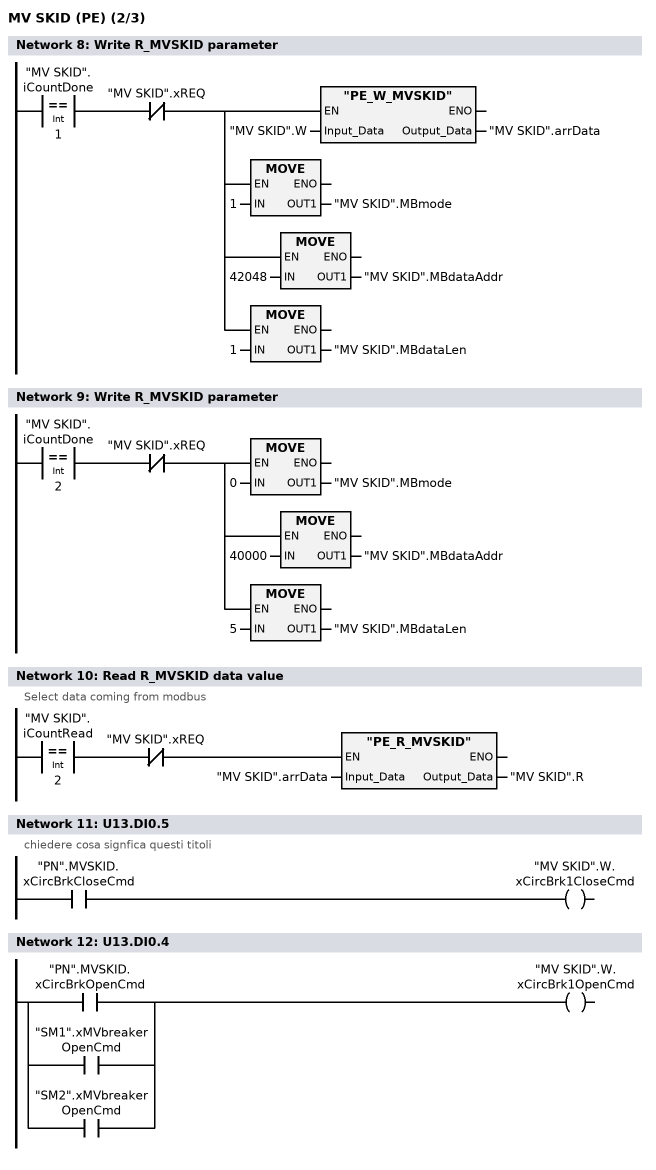
   RUNG wire#powerrail
      { S7_Templates := "SrcType := Int" } EQ_Contact(in1 := "MV SKID".iCountDone, in2 := 1)
      I_Contact( "MV SKID".xREQ )
      wire#w1
      "PE_W_MVSKID"(Input_Data := "MV SKID".W, Output_Data => "MV SKID".arrData)
   END_RUNG
   RUNG wire#w1
      Move(in := 1, out1 => "MV SKID".MBmode)
   END_RUNG
   RUNG wire#w1
      Move(in := 42048, out1 => "MV SKID".MBdataAddr)
   END_RUNG
   RUNG wire#w1
      Move(in := 1, out1 => "MV SKID".MBdataLen)
   END_RUNG
   // the same network as SCL:
   #_w1 := ("MV SKID".iCountDone = 1) AND NOT "MV SKID".xREQ;
   IF #_w1 THEN
       "PE_W_MVSKID"(Input_Data := "MV SKID".W, Output_Data => "MV SKID".arrData);
       "MV SKID".MBmode := 1;
       "MV SKID".MBdataAddr := 42048;
       "MV SKID".MBdataLen := 1;
   END_IF;
END_REGION

REGION Network 9: Write R_MVSKID parameter
   RUNG wire#powerrail
      { S7_Templates := "SrcType := Int" } EQ_Contact(in1 := "MV SKID".iCountDone, in2 := 2)
      I_Contact( "MV SKID".xREQ )
      wire#w1
      Move(in := 0, out1 => "MV SKID".MBmode)
   END_RUNG
   RUNG wire#w1
      Move(in := 40000, out1 => "MV SKID".MBdataAddr)
   END_RUNG
   RUNG wire#w1
      Move(in := 5, out1 => "MV SKID".MBdataLen)
   END_RUNG
   // the same network as SCL:
   IF ("MV SKID".iCountDone = 2) AND NOT "MV SKID".xREQ THEN
       "MV SKID".MBmode := 0;
       "MV SKID".MBdataAddr := 40000;
       "MV SKID".MBdataLen := 5;
   END_IF;
END_REGION

REGION Network 10: Read R_MVSKID data value
   // Select data coming from modbus
   RUNG wire#powerrail
      { S7_Templates := "SrcType := Int" } EQ_Contact(in1 := "MV SKID".iCountRead, in2 := 2)
      I_Contact( "MV SKID".xREQ )
      "PE_R_MVSKID"(Input_Data := "MV SKID".arrData, Output_Data => "MV SKID".R)
   END_RUNG
   // the same network as SCL:
   IF ("MV SKID".iCountRead = 2) AND NOT "MV SKID".xREQ THEN
       "PE_R_MVSKID"(Input_Data := "MV SKID".arrData, Output_Data => "MV SKID".R);
   END_IF;
END_REGION

REGION Network 11: U13.DI0.5
   // chiedere cosa signfica questi titoli
   RUNG wire#powerrail
      Contact( "PN".MVSKID.xCircBrkCloseCmd )
      Coil( "MV SKID".W.xCircBrk1CloseCmd )
   END_RUNG
   // the same network as SCL:
   "MV SKID".W.xCircBrk1CloseCmd := "PN".MVSKID.xCircBrkCloseCmd;
END_REGION

REGION Network 12: U13.DI0.4
   RUNG wire#powerrail
      Contact( "PN".MVSKID.xCircBrkOpenCmd )
      wire#w1
      Coil( "MV SKID".W.xCircBrk1OpenCmd )
   END_RUNG
   RUNG wire#powerrail
      Contact( "SM1".xMVbreakerOpenCmd )
   END_RUNG wire#w1
   RUNG wire#powerrail
      Contact( "SM2".xMVbreakerOpenCmd )
   END_RUNG wire#w1
   // the same network as SCL:
   "MV SKID".W.xCircBrk1OpenCmd := "PN".MVSKID.xCircBrkOpenCmd OR "SM1".xMVbreakerOpenCmd OR "SM2".xMVbreakerOpenCmd;
END_REGION

REGION Network 13: MV SKID Fault
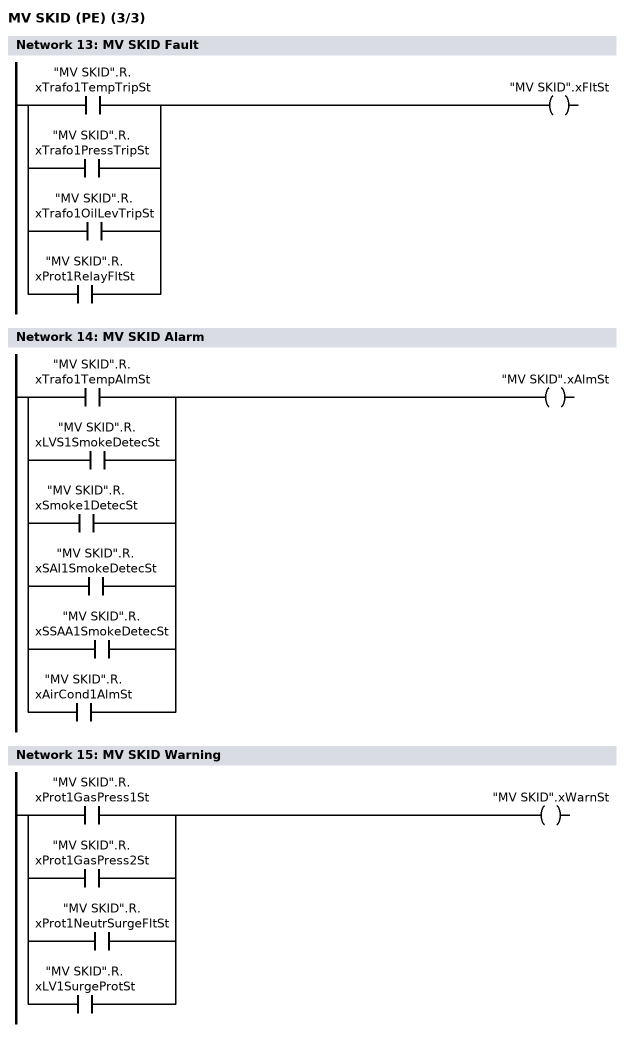
   RUNG wire#powerrail
      Contact( "MV SKID".R.xTrafo1TempTripSt )
      wire#w1
      Coil( "MV SKID".xFltSt )
   END_RUNG
   RUNG wire#powerrail
      Contact( "MV SKID".R.xTrafo1PressTripSt )
   END_RUNG wire#w1
   RUNG wire#powerrail
      Contact( "MV SKID".R.xTrafo1OilLevTripSt )
   END_RUNG wire#w1
   RUNG wire#powerrail
      Contact( "MV SKID".R.xProt1RelayFltSt )
   END_RUNG wire#w1
   // the same network as SCL:
   "MV SKID".xFltSt := "MV SKID".R.xTrafo1TempTripSt OR "MV SKID".R.xTrafo1PressTripSt OR "MV SKID".R.xTrafo1OilLevTripSt OR "MV SKID".R.xProt1RelayFltSt;
END_REGION

REGION Network 14: MV SKID Alarm
   RUNG wire#powerrail
      Contact( "MV SKID".R.xTrafo1TempAlmSt )
      wire#w1
      Coil( "MV SKID".xAlmSt )
   END_RUNG
   RUNG wire#powerrail
      Contact( "MV SKID".R.xLVS1SmokeDetecSt )
   END_RUNG wire#w1
   RUNG wire#powerrail
      Contact( "MV SKID".R.xSmoke1DetecSt )
   END_RUNG wire#w1
   RUNG wire#powerrail
      Contact( "MV SKID".R.xSAI1SmokeDetecSt )
   END_RUNG wire#w1
   RUNG wire#powerrail
      Contact( "MV SKID".R.xSSAA1SmokeDetecSt )
   END_RUNG wire#w1
   RUNG wire#powerrail
      Contact( "MV SKID".R.xAirCond1AlmSt )
   END_RUNG wire#w1
   // the same network as SCL:
   "MV SKID".xAlmSt := "MV SKID".R.xTrafo1TempAlmSt OR "MV SKID".R.xLVS1SmokeDetecSt OR "MV SKID".R.xSmoke1DetecSt OR "MV SKID".R.xSAI1SmokeDetecSt OR "MV SKID".R.xSSAA1SmokeDetecSt OR "MV SKID".R.xAirCond1AlmSt;
END_REGION

REGION Network 15: MV SKID Warning
   RUNG wire#powerrail
      Contact( "MV SKID".R.xProt1GasPress1St )
      wire#w1
      Coil( "MV SKID".xWarnSt )
   END_RUNG
   RUNG wire#powerrail
      Contact( "MV SKID".R.xProt1GasPress2St )
   END_RUNG wire#w1
   RUNG wire#powerrail
      Contact( "MV SKID".R.xProt1NeutrSurgeFltSt )
   END_RUNG wire#w1
   RUNG wire#powerrail
      Contact( "MV SKID".R.xLV1SurgeProtSt )
   END_RUNG wire#w1
   // the same network as SCL:
   "MV SKID".xWarnSt := "MV SKID".R.xProt1GasPress1St OR "MV SKID".R.xProt1GasPress2St OR "MV SKID".R.xProt1NeutrSurgeFltSt OR "MV SKID".R.xLV1SurgeProtSt;
END_REGION

REGION Network 16 (SCL): MV SKID Line Disconnector & Breaker Status
   "MV SKID".wLine1DiscSt.%X0 := "MV SKID".R.xLine1DiscOpenSt;
   "MV SKID".wLine1DiscSt.%X1 := "MV SKID".R.xLine1DiscCloseSt;
   "MV SKID".wLine1DiscSt.%X2 := "MV SKID".R.xLine1GndCloseSt;

   "MV SKID".wLine2DiscSt.%X0 := "MV SKID".R.xLine2DiscOpenSt;
   "MV SKID".wLine2DiscSt.%X1 := "MV SKID".R.xLine2DiscCloseSt;
   "MV SKID".wLine2DiscSt.%X2 := "MV SKID".R.xLine2GndCloseSt;

   "MV SKID".wProt1DiscSt.%X0 := "MV SKID".R.xProt1DiscOpenSt;
   "MV SKID".wProt1DiscSt.%X1 := "MV SKID".R.xProt1DiscCloseSt;
   "MV SKID".wProt1DiscSt.%X2 := "MV SKID".R.xProt1GndCloseSt;

   "MV SKID".wProt1CircBrkSt.%X0 := "MV SKID".R.xProt1CircBrkOpenSt;
   "MV SKID".wProt1CircBrkSt.%X1 := "MV SKID".R.xProt1CircBrkCloseSt;
END_REGION
END_FUNCTION

FUNCTION "PE_W_MVSKID" : Void
{ S7_Optimized_Access := 'TRUE' }
VERSION : 0.1
   VAR_INPUT 
      Input_Data : "W_MV";
   END_VAR

   VAR_OUTPUT 
      Output_Data : Array[1..125] of Word;
   END_VAR


BEGIN
	REGION
	    // 2022/01/24
	END_REGION
	
	REGION
	    
	    #Output_Data[1].%X0 := #Input_Data.xCircBrk1OpenCmd;
	    #Output_Data[1].%X1 := #Input_Data.xCircBrk1CloseCmd;
	    #Output_Data[1].%X2 := #Input_Data.xLVCircBrk1OpenCmd;
	    #Output_Data[1].%X3 := #Input_Data.xLVCircBrk1CloseCmd;
	    #Output_Data[1].%X4 := #Input_Data.xCircBrk2OpenCmd;
	    #Output_Data[1].%X5 := #Input_Data.xCircBrk2CloseCmd;
	    #Output_Data[1].%X6 := #Input_Data.xLVCircBrk2OpenCmd;
	    #Output_Data[1].%X7 := #Input_Data.xLVCircBrk2CloseCmd;
	    
	END_REGION
END_FUNCTION

FUNCTION "PE_R_MVSKID" : Void
{ S7_Optimized_Access := 'TRUE' }
VERSION : 0.1
   VAR_INPUT 
      Input_Data : Array[1..125] of Word;
   END_VAR

   VAR_OUTPUT 
      Output_Data : "R_MV";
   END_VAR


BEGIN
	REGION
	    // 2022/01/24
	END_REGION
	
	REGION
	    
	    #Output_Data.xTrafo1TempTripSt      := #Input_Data[1].%X0;
	    #Output_Data.xTrafo1TempAlmSt       := #Input_Data[1].%X1;
	    #Output_Data.xTrafo1PressTripSt     := #Input_Data[1].%X2;
	    #Output_Data.xTrafo1OilLevTripSt    := #Input_Data[1].%X3;
	    #Output_Data.xLine1DiscOpenSt       := #Input_Data[1].%X4;
	    #Output_Data.xLine1DiscCloseSt      := #Input_Data[1].%X5;
	    #Output_Data.xLine1GndCloseSt       := #Input_Data[1].%X6;
	    #Output_Data.xProt1GasPress1St      := #Input_Data[1].%X7;
	    
	    #Output_Data.xLine2DiscOpenSt       := #Input_Data[1].%X8;
	    #Output_Data.xLine2DiscCloseSt      := #Input_Data[1].%X9;
	    #Output_Data.xLine2GndCloseSt       := #Input_Data[1].%X10;
	    #Output_Data.xProt1DiscCloseSt      := #Input_Data[1].%X11;
	    #Output_Data.xProt1DiscOpenSt       := #Input_Data[1].%X12;
	    #Output_Data.xProt1GndCloseSt       := #Input_Data[1].%X13;
	    #Output_Data.xProt1CircBrkOpenSt    := #Input_Data[1].%X14;
	    #Output_Data.xProt1CircBrkCloseSt   := #Input_Data[1].%X15;
	    
	    #Output_Data.xProt1RelayFltSt       := #Input_Data[2].%X0;
	    #Output_Data.xLV1SurgeProtSt        := #Input_Data[2].%X1;
	    #Output_Data.xSpring1ChargeSt       := #Input_Data[2].%X2;
	    #Output_Data.xProt1GasPress2St      := #Input_Data[2].%X3;
	    #Output_Data.xBackfeedtrakers1St    := #Input_Data[2].%X4;
	    #Output_Data.xProt1NeutrSurgeFltSt  := #Input_Data[2].%X5;
	    #Output_Data.xLVS1SmokeDetecSt       := #Input_Data[2].%X6;
	    #Output_Data.xSmoke1DetecSt         := #Input_Data[2].%X7;
	    
	    #Output_Data.xSAI1SmokeDetecSt      := #Input_Data[2].%X8;
	    #Output_Data.xSSAA1SmokeDetecSt     := #Input_Data[2].%X9;
	    #Output_Data.xAirCond1AlmSt         := #Input_Data[2].%X10;
	    #Output_Data.xAcBrkHENK1OpenSt      := #Input_Data[2].%X11;
	    #Output_Data.xAcBrkHENK1CloseSt     := #Input_Data[2].%X12;
	    #Output_Data.xTrafo2TempTripSt      := #Input_Data[2].%X13;
	    #Output_Data.xTrafo2TempAlmSt       := #Input_Data[2].%X14;
	    #Output_Data.xTrafo2PressTripSt     := #Input_Data[2].%X15;
	    
	    #Output_Data.xTrafo2OilLevTripSt    := #Input_Data[3].%X0;
	    #Output_Data.xProt2DiscCloseSt      := #Input_Data[3].%X1;
	    #Output_Data.xProt2DiscOpenSt       := #Input_Data[3].%X2;
	    #Output_Data.xProt2GndCloseSt       := #Input_Data[3].%X3;
	    #Output_Data.xProt2CircBrkOpenSt    := #Input_Data[3].%X4;
	    #Output_Data.xProt2CircBrkCloseSt   := #Input_Data[3].%X5;
	    #Output_Data.xProt2NCWatchdogSt     := #Input_Data[3].%X6;
	    #Output_Data.xLV2SurgeProtSt        := #Input_Data[3].%X7;
	    
	    #Output_Data.xSpring2ChargeSt       := #Input_Data[3].%X8;
	    #Output_Data.xAcBrkHENK2OpenSt      := #Input_Data[3].%X9;
	    #Output_Data.xAcBrkHENK2CloseSt     := #Input_Data[3].%X10;
	    #Output_Data.xBackfeedtrakers2St    := #Input_Data[3].%X11;
	    #Output_Data.xProt2NeutrSurgeSt     := #Input_Data[3].%X12;
	    #Output_Data.xSAI2SmokeDetecSt      := #Input_Data[3].%X13;
	    #Output_Data.xSSAA2SmokeDetecSt     := #Input_Data[3].%X14;
	    #Output_Data.xAirCond2AlmSt         := #Input_Data[3].%X15;
	    
	    #Output_Data.rPT100Trafo1St         := INT_TO_REAL(WORD_TO_INT(#Input_Data[4]))/10.0;
	    #Output_Data.rPT100Trafo2St         := INT_TO_REAL(WORD_TO_INT(#Input_Data[5]))/10.0;
	    
	END_REGION
END_FUNCTION

FUNCTION "PCS1 Faults" : Void   // FC43, LAD
{ S7_Optimized_Access := 'TRUE' }
VERSION : 0.1
// stored: AutoNumber false, IsIECCheckEnabled false, SetENOAutomatically false, UDAEnableTagReadback false
   VAR_TEMP
      wMF1 : Word;
      wMF2 : Word;
      wMF3 : Word;
      wMF4 : Word;
      wMW1 : Word;
      wMW2 : Word;
      wMW3 : Word;
      wMW4 : Word;
   END_VAR
   VAR_TEMP   // added for the SCL form of the ladder/FBD networks
      _w1 : Bool;
      _w2 : Bool;
      _w3 : Bool;
      _w4 : Bool;
   END_VAR
BEGIN

REGION Network 1: Split Inverter fault & warning and Module number
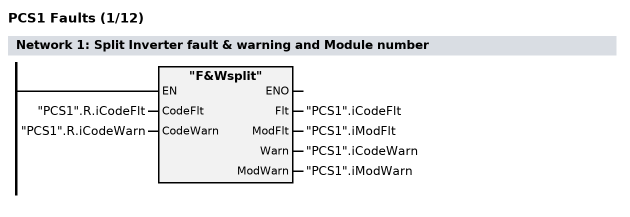
   RUNG wire#powerrail
      "F&Wsplit"(CodeFlt := "PCS1".R.iCodeFlt, CodeWarn := "PCS1".R.iCodeWarn, Flt => "PCS1".iCodeFlt, ModFlt => "PCS1".iModFlt, Warn => "PCS1".iCodeWarn, ModWarn => "PCS1".iModWarn)
   END_RUNG
   // the same network as SCL:
   "F&Wsplit"(CodeFlt := "PCS1".R.iCodeFlt,
              CodeWarn := "PCS1".R.iCodeWarn,
              Flt => "PCS1".iCodeFlt,
              ModFlt => "PCS1".iModFlt,
              Warn => "PCS1".iCodeWarn,
              ModWarn => "PCS1".iModWarn);
END_REGION

REGION Network 2: Inverter Faults
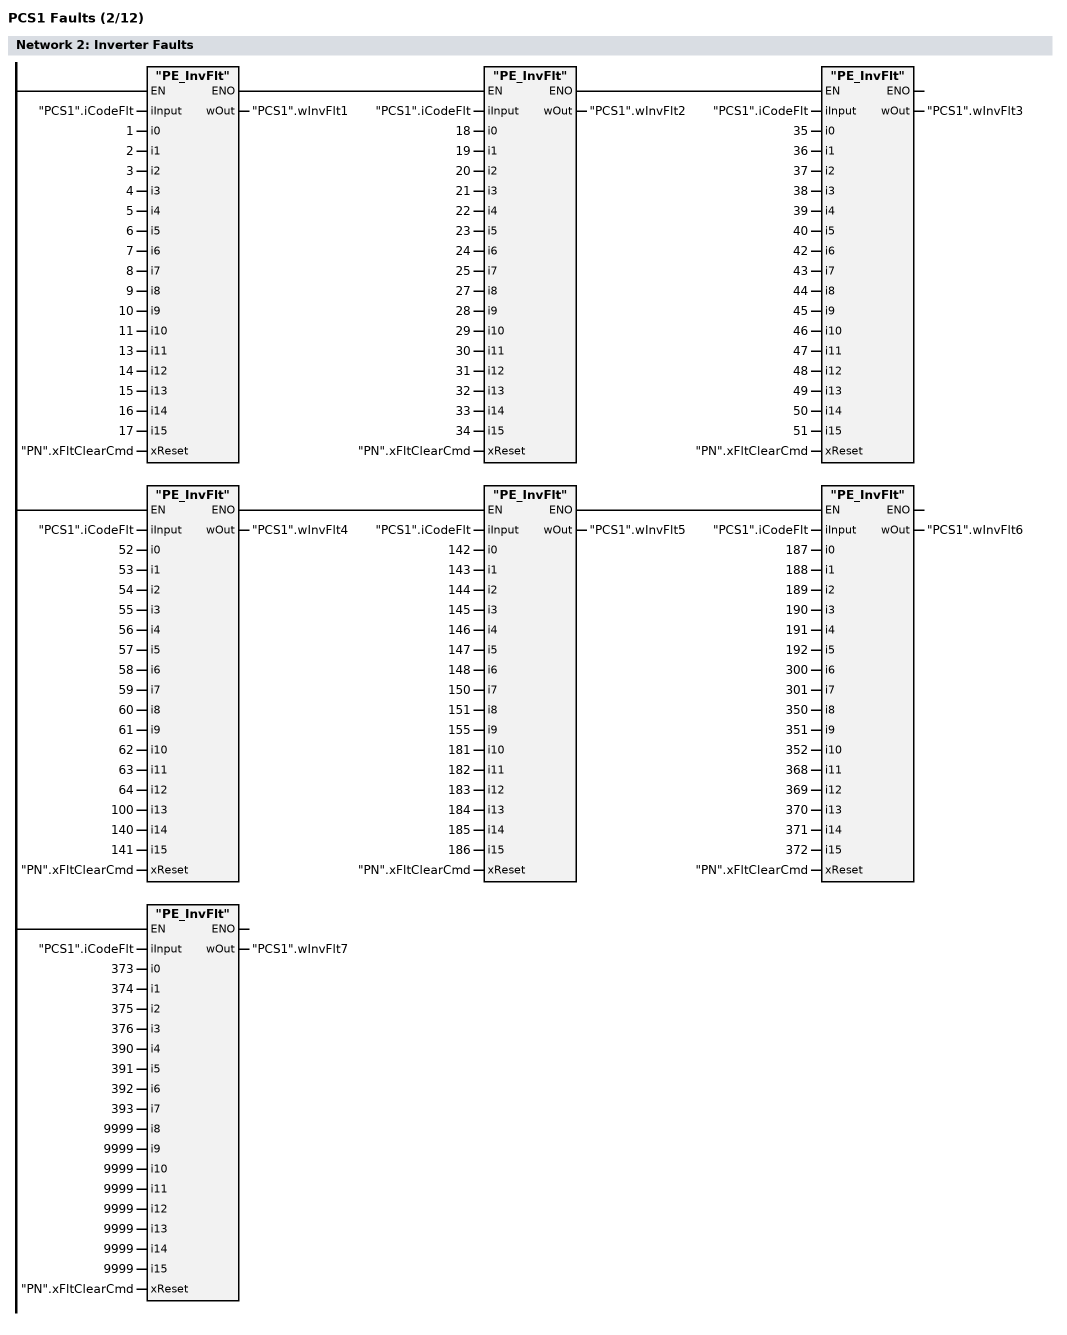
   RUNG wire#powerrail
      "PE_InvFlt"(iInput := "PCS1".iCodeFlt, i0 := 1, i1 := 2, i2 := 3, i3 := 4, i4 := 5, i5 := 6, i6 := 7, i7 := 8, i8 := 9, i9 := 10, i10 := 11, i11 := 13, i12 := 14, i13 := 15, i14 := 16, i15 := 17, xReset := "PN".xFltClearCmd, wOut => "PCS1".wInvFlt1)
      "PE_InvFlt"(iInput := "PCS1".iCodeFlt, i0 := 18, i1 := 19, i2 := 20, i3 := 21, i4 := 22, i5 := 23, i6 := 24, i7 := 25, i8 := 27, i9 := 28, i10 := 29, i11 := 30, i12 := 31, i13 := 32, i14 := 33, i15 := 34, xReset := "PN".xFltClearCmd, wOut => "PCS1".wInvFlt2)
      "PE_InvFlt"(iInput := "PCS1".iCodeFlt, i0 := 35, i1 := 36, i2 := 37, i3 := 38, i4 := 39, i5 := 40, i6 := 42, i7 := 43, i8 := 44, i9 := 45, i10 := 46, i11 := 47, i12 := 48, i13 := 49, i14 := 50, i15 := 51, xReset := "PN".xFltClearCmd, wOut => "PCS1".wInvFlt3)
   END_RUNG
   RUNG wire#powerrail
      "PE_InvFlt"(iInput := "PCS1".iCodeFlt, i0 := 52, i1 := 53, i2 := 54, i3 := 55, i4 := 56, i5 := 57, i6 := 58, i7 := 59, i8 := 60, i9 := 61, i10 := 62, i11 := 63, i12 := 64, i13 := 100, i14 := 140, i15 := 141, xReset := "PN".xFltClearCmd, wOut => "PCS1".wInvFlt4)
      "PE_InvFlt"(iInput := "PCS1".iCodeFlt, i0 := 142, i1 := 143, i2 := 144, i3 := 145, i4 := 146, i5 := 147, i6 := 148, i7 := 150, i8 := 151, i9 := 155, i10 := 181, i11 := 182, i12 := 183, i13 := 184, i14 := 185, i15 := 186, xReset := "PN".xFltClearCmd, wOut => "PCS1".wInvFlt5)
      "PE_InvFlt"(iInput := "PCS1".iCodeFlt, i0 := 187, i1 := 188, i2 := 189, i3 := 190, i4 := 191, i5 := 192, i6 := 300, i7 := 301, i8 := 350, i9 := 351, i10 := 352, i11 := 368, i12 := 369, i13 := 370, i14 := 371, i15 := 372, xReset := "PN".xFltClearCmd, wOut => "PCS1".wInvFlt6)
   END_RUNG
   RUNG wire#powerrail
      "PE_InvFlt"(iInput := "PCS1".iCodeFlt, i0 := 373, i1 := 374, i2 := 375, i3 := 376, i4 := 390, i5 := 391, i6 := 392, i7 := 393, i8 := 9999, i9 := 9999, i10 := 9999, i11 := 9999, i12 := 9999, i13 := 9999, i14 := 9999, i15 := 9999, xReset := "PN".xFltClearCmd, wOut => "PCS1".wInvFlt7)
   END_RUNG
   // the same network as SCL:
   "PE_InvFlt"(iInput := "PCS1".iCodeFlt,
               i0 := 1,
               i1 := 2,
               i2 := 3,
               i3 := 4,
               i4 := 5,
               i5 := 6,
               i6 := 7,
               i7 := 8,
               i8 := 9,
               i9 := 10,
               i10 := 11,
               i11 := 13,
               i12 := 14,
               i13 := 15,
               i14 := 16,
               i15 := 17,
               xReset := "PN".xFltClearCmd,
               wOut => "PCS1".wInvFlt1,
               ENO => #_w1);
   "PE_InvFlt"(EN := #_w1,
               iInput := "PCS1".iCodeFlt,
               i0 := 18,
               i1 := 19,
               i2 := 20,
               i3 := 21,
               i4 := 22,
               i5 := 23,
               i6 := 24,
               i7 := 25,
               i8 := 27,
               i9 := 28,
               i10 := 29,
               i11 := 30,
               i12 := 31,
               i13 := 32,
               i14 := 33,
               i15 := 34,
               xReset := "PN".xFltClearCmd,
               wOut => "PCS1".wInvFlt2,
               ENO => #_w2);
   IF #_w2 THEN
       "PE_InvFlt"(iInput := "PCS1".iCodeFlt,
                   i0 := 35,
                   i1 := 36,
                   i2 := 37,
                   i3 := 38,
                   i4 := 39,
                   i5 := 40,
                   i6 := 42,
                   i7 := 43,
                   i8 := 44,
                   i9 := 45,
                   i10 := 46,
                   i11 := 47,
                   i12 := 48,
                   i13 := 49,
                   i14 := 50,
                   i15 := 51,
                   xReset := "PN".xFltClearCmd,
                   wOut => "PCS1".wInvFlt3);
   END_IF;
   "PE_InvFlt"(iInput := "PCS1".iCodeFlt,
               i0 := 52,
               i1 := 53,
               i2 := 54,
               i3 := 55,
               i4 := 56,
               i5 := 57,
               i6 := 58,
               i7 := 59,
               i8 := 60,
               i9 := 61,
               i10 := 62,
               i11 := 63,
               i12 := 64,
               i13 := 100,
               i14 := 140,
               i15 := 141,
               xReset := "PN".xFltClearCmd,
               wOut => "PCS1".wInvFlt4,
               ENO => #_w3);
   "PE_InvFlt"(EN := #_w3,
               iInput := "PCS1".iCodeFlt,
               i0 := 142,
               i1 := 143,
               i2 := 144,
               i3 := 145,
               i4 := 146,
               i5 := 147,
               i6 := 148,
               i7 := 150,
               i8 := 151,
               i9 := 155,
               i10 := 181,
               i11 := 182,
               i12 := 183,
               i13 := 184,
               i14 := 185,
               i15 := 186,
               xReset := "PN".xFltClearCmd,
               wOut => "PCS1".wInvFlt5,
               ENO => #_w4);
   IF #_w4 THEN
       "PE_InvFlt"(iInput := "PCS1".iCodeFlt,
                   i0 := 187,
                   i1 := 188,
                   i2 := 189,
                   i3 := 190,
                   i4 := 191,
                   i5 := 192,
                   i6 := 300,
                   i7 := 301,
                   i8 := 350,
                   i9 := 351,
                   i10 := 352,
                   i11 := 368,
                   i12 := 369,
                   i13 := 370,
                   i14 := 371,
                   i15 := 372,
                   xReset := "PN".xFltClearCmd,
                   wOut => "PCS1".wInvFlt6);
   END_IF;
   "PE_InvFlt"(iInput := "PCS1".iCodeFlt,
               i0 := 373,
               i1 := 374,
               i2 := 375,
               i3 := 376,
               i4 := 390,
               i5 := 391,
               i6 := 392,
               i7 := 393,
               i8 := 9999,
               i9 := 9999,
               i10 := 9999,
               i11 := 9999,
               i12 := 9999,
               i13 := 9999,
               i14 := 9999,
               i15 := 9999,
               xReset := "PN".xFltClearCmd,
               wOut => "PCS1".wInvFlt7);
END_REGION

REGION Network 3: Inverter Warning
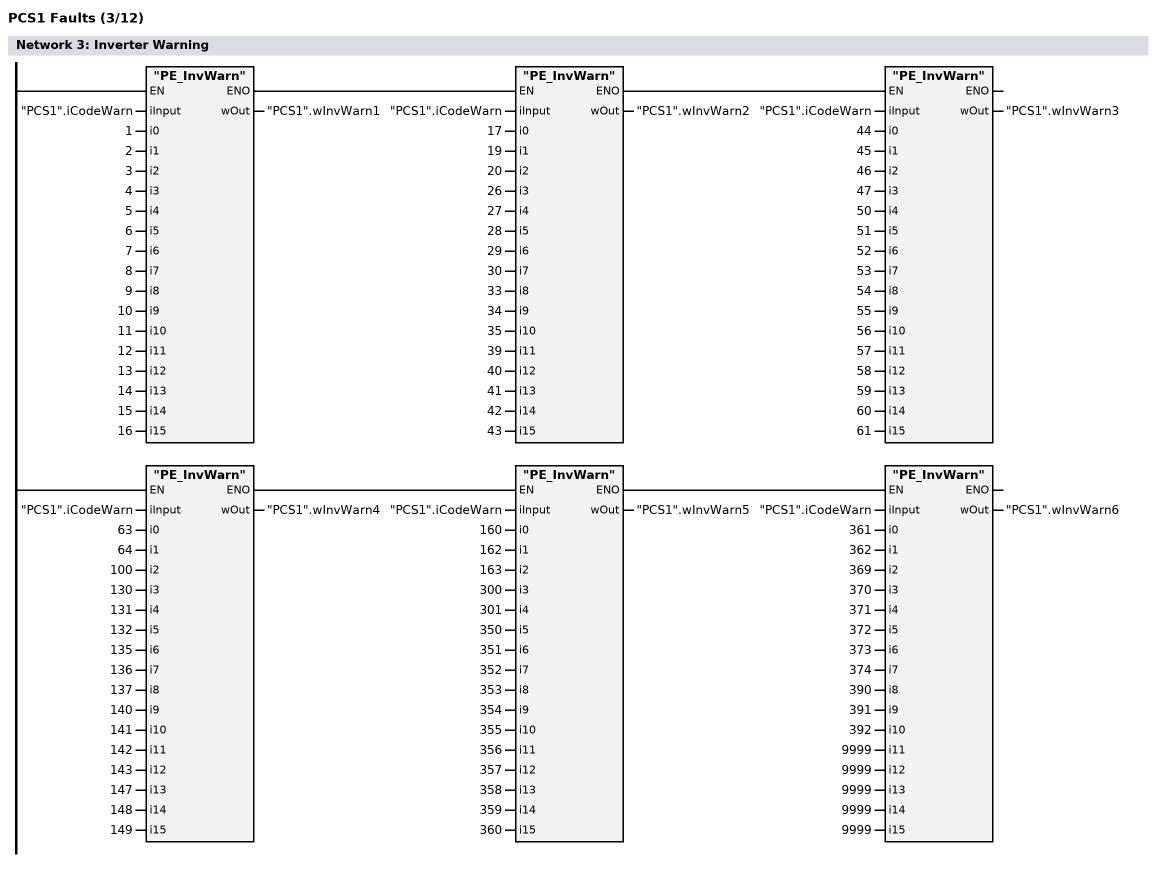
   RUNG wire#powerrail
      "PE_InvWarn"(iInput := "PCS1".iCodeWarn, i0 := 1, i1 := 2, i2 := 3, i3 := 4, i4 := 5, i5 := 6, i6 := 7, i7 := 8, i8 := 9, i9 := 10, i10 := 11, i11 := 12, i12 := 13, i13 := 14, i14 := 15, i15 := 16, wOut => "PCS1".wInvWarn1)
      "PE_InvWarn"(iInput := "PCS1".iCodeWarn, i0 := 17, i1 := 19, i2 := 20, i3 := 26, i4 := 27, i5 := 28, i6 := 29, i7 := 30, i8 := 33, i9 := 34, i10 := 35, i11 := 39, i12 := 40, i13 := 41, i14 := 42, i15 := 43, wOut => "PCS1".wInvWarn2)
      "PE_InvWarn"(iInput := "PCS1".iCodeWarn, i0 := 44, i1 := 45, i2 := 46, i3 := 47, i4 := 50, i5 := 51, i6 := 52, i7 := 53, i8 := 54, i9 := 55, i10 := 56, i11 := 57, i12 := 58, i13 := 59, i14 := 60, i15 := 61, wOut => "PCS1".wInvWarn3)
   END_RUNG
   RUNG wire#powerrail
      "PE_InvWarn"(iInput := "PCS1".iCodeWarn, i0 := 63, i1 := 64, i2 := 100, i3 := 130, i4 := 131, i5 := 132, i6 := 135, i7 := 136, i8 := 137, i9 := 140, i10 := 141, i11 := 142, i12 := 143, i13 := 147, i14 := 148, i15 := 149, wOut => "PCS1".wInvWarn4)
      "PE_InvWarn"(iInput := "PCS1".iCodeWarn, i0 := 160, i1 := 162, i2 := 163, i3 := 300, i4 := 301, i5 := 350, i6 := 351, i7 := 352, i8 := 353, i9 := 354, i10 := 355, i11 := 356, i12 := 357, i13 := 358, i14 := 359, i15 := 360, wOut => "PCS1".wInvWarn5)
      "PE_InvWarn"(iInput := "PCS1".iCodeWarn, i0 := 361, i1 := 362, i2 := 369, i3 := 370, i4 := 371, i5 := 372, i6 := 373, i7 := 374, i8 := 390, i9 := 391, i10 := 392, i11 := 9999, i12 := 9999, i13 := 9999, i14 := 9999, i15 := 9999, wOut => "PCS1".wInvWarn6)
   END_RUNG
   // the same network as SCL:
   "PE_InvWarn"(iInput := "PCS1".iCodeWarn,
                i0 := 1,
                i1 := 2,
                i2 := 3,
                i3 := 4,
                i4 := 5,
                i5 := 6,
                i6 := 7,
                i7 := 8,
                i8 := 9,
                i9 := 10,
                i10 := 11,
                i11 := 12,
                i12 := 13,
                i13 := 14,
                i14 := 15,
                i15 := 16,
                wOut => "PCS1".wInvWarn1,
                ENO => #_w1);
   "PE_InvWarn"(EN := #_w1,
                iInput := "PCS1".iCodeWarn,
                i0 := 17,
                i1 := 19,
                i2 := 20,
                i3 := 26,
                i4 := 27,
                i5 := 28,
                i6 := 29,
                i7 := 30,
                i8 := 33,
                i9 := 34,
                i10 := 35,
                i11 := 39,
                i12 := 40,
                i13 := 41,
                i14 := 42,
                i15 := 43,
                wOut => "PCS1".wInvWarn2,
                ENO => #_w2);
   IF #_w2 THEN
       "PE_InvWarn"(iInput := "PCS1".iCodeWarn,
                    i0 := 44,
                    i1 := 45,
                    i2 := 46,
                    i3 := 47,
                    i4 := 50,
                    i5 := 51,
                    i6 := 52,
                    i7 := 53,
                    i8 := 54,
                    i9 := 55,
                    i10 := 56,
                    i11 := 57,
                    i12 := 58,
                    i13 := 59,
                    i14 := 60,
                    i15 := 61,
                    wOut => "PCS1".wInvWarn3);
   END_IF;
   "PE_InvWarn"(iInput := "PCS1".iCodeWarn,
                i0 := 63,
                i1 := 64,
                i2 := 100,
                i3 := 130,
                i4 := 131,
                i5 := 132,
                i6 := 135,
                i7 := 136,
                i8 := 137,
                i9 := 140,
                i10 := 141,
                i11 := 142,
                i12 := 143,
                i13 := 147,
                i14 := 148,
                i15 := 149,
                wOut => "PCS1".wInvWarn4,
                ENO => #_w3);
   "PE_InvWarn"(EN := #_w3,
                iInput := "PCS1".iCodeWarn,
                i0 := 160,
                i1 := 162,
                i2 := 163,
                i3 := 300,
                i4 := 301,
                i5 := 350,
                i6 := 351,
                i7 := 352,
                i8 := 353,
                i9 := 354,
                i10 := 355,
                i11 := 356,
                i12 := 357,
                i13 := 358,
                i14 := 359,
                i15 := 360,
                wOut => "PCS1".wInvWarn5,
                ENO => #_w4);
   IF #_w4 THEN
       "PE_InvWarn"(iInput := "PCS1".iCodeWarn,
                    i0 := 361,
                    i1 := 362,
                    i2 := 369,
                    i3 := 370,
                    i4 := 371,
                    i5 := 372,
                    i6 := 373,
                    i7 := 374,
                    i8 := 390,
                    i9 := 391,
                    i10 := 392,
                    i11 := 9999,
                    i12 := 9999,
                    i13 := 9999,
                    i14 := 9999,
                    i15 := 9999,
                    wOut => "PCS1".wInvWarn6);
   END_IF;
END_REGION

REGION Network 4: Module Faults
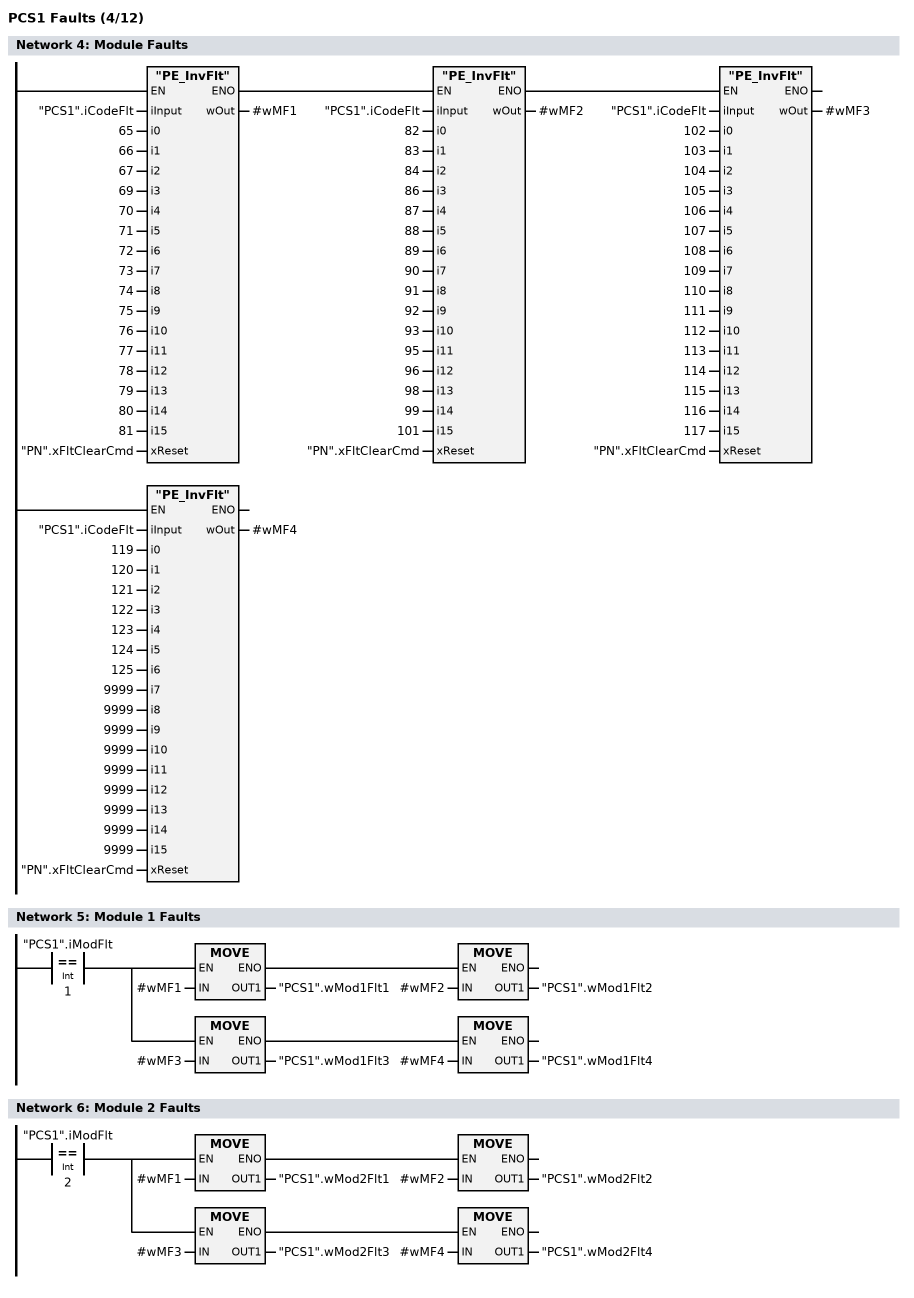
   RUNG wire#powerrail
      "PE_InvFlt"(iInput := "PCS1".iCodeFlt, i0 := 65, i1 := 66, i2 := 67, i3 := 69, i4 := 70, i5 := 71, i6 := 72, i7 := 73, i8 := 74, i9 := 75, i10 := 76, i11 := 77, i12 := 78, i13 := 79, i14 := 80, i15 := 81, xReset := "PN".xFltClearCmd, wOut => #wMF1)
      "PE_InvFlt"(iInput := "PCS1".iCodeFlt, i0 := 82, i1 := 83, i2 := 84, i3 := 86, i4 := 87, i5 := 88, i6 := 89, i7 := 90, i8 := 91, i9 := 92, i10 := 93, i11 := 95, i12 := 96, i13 := 98, i14 := 99, i15 := 101, xReset := "PN".xFltClearCmd, wOut => #wMF2)
      "PE_InvFlt"(iInput := "PCS1".iCodeFlt, i0 := 102, i1 := 103, i2 := 104, i3 := 105, i4 := 106, i5 := 107, i6 := 108, i7 := 109, i8 := 110, i9 := 111, i10 := 112, i11 := 113, i12 := 114, i13 := 115, i14 := 116, i15 := 117, xReset := "PN".xFltClearCmd, wOut => #wMF3)
   END_RUNG
   RUNG wire#powerrail
      "PE_InvFlt"(iInput := "PCS1".iCodeFlt, i0 := 119, i1 := 120, i2 := 121, i3 := 122, i4 := 123, i5 := 124, i6 := 125, i7 := 9999, i8 := 9999, i9 := 9999, i10 := 9999, i11 := 9999, i12 := 9999, i13 := 9999, i14 := 9999, i15 := 9999, xReset := "PN".xFltClearCmd, wOut => #wMF4)
   END_RUNG
   // the same network as SCL:
   "PE_InvFlt"(iInput := "PCS1".iCodeFlt,
               i0 := 65,
               i1 := 66,
               i2 := 67,
               i3 := 69,
               i4 := 70,
               i5 := 71,
               i6 := 72,
               i7 := 73,
               i8 := 74,
               i9 := 75,
               i10 := 76,
               i11 := 77,
               i12 := 78,
               i13 := 79,
               i14 := 80,
               i15 := 81,
               xReset := "PN".xFltClearCmd,
               wOut => #wMF1,
               ENO => #_w1);
   "PE_InvFlt"(EN := #_w1,
               iInput := "PCS1".iCodeFlt,
               i0 := 82,
               i1 := 83,
               i2 := 84,
               i3 := 86,
               i4 := 87,
               i5 := 88,
               i6 := 89,
               i7 := 90,
               i8 := 91,
               i9 := 92,
               i10 := 93,
               i11 := 95,
               i12 := 96,
               i13 := 98,
               i14 := 99,
               i15 := 101,
               xReset := "PN".xFltClearCmd,
               wOut => #wMF2,
               ENO => #_w2);
   IF #_w2 THEN
       "PE_InvFlt"(iInput := "PCS1".iCodeFlt,
                   i0 := 102,
                   i1 := 103,
                   i2 := 104,
                   i3 := 105,
                   i4 := 106,
                   i5 := 107,
                   i6 := 108,
                   i7 := 109,
                   i8 := 110,
                   i9 := 111,
                   i10 := 112,
                   i11 := 113,
                   i12 := 114,
                   i13 := 115,
                   i14 := 116,
                   i15 := 117,
                   xReset := "PN".xFltClearCmd,
                   wOut => #wMF3);
   END_IF;
   "PE_InvFlt"(iInput := "PCS1".iCodeFlt,
               i0 := 119,
               i1 := 120,
               i2 := 121,
               i3 := 122,
               i4 := 123,
               i5 := 124,
               i6 := 125,
               i7 := 9999,
               i8 := 9999,
               i9 := 9999,
               i10 := 9999,
               i11 := 9999,
               i12 := 9999,
               i13 := 9999,
               i14 := 9999,
               i15 := 9999,
               xReset := "PN".xFltClearCmd,
               wOut => #wMF4);
END_REGION

REGION Network 5: Module 1 Faults
   RUNG wire#powerrail
      { S7_Templates := "SrcType := Int" } EQ_Contact(in1 := "PCS1".iModFlt, in2 := 1)
      wire#w1
      Move(in := #wMF1, out1 => "PCS1".wMod1Flt1)
      Move(in := #wMF2, out1 => "PCS1".wMod1Flt2)
   END_RUNG
   RUNG wire#w1
      Move(in := #wMF3, out1 => "PCS1".wMod1Flt3)
      Move(in := #wMF4, out1 => "PCS1".wMod1Flt4)
   END_RUNG
   // the same network as SCL:
   IF "PCS1".iModFlt = 1 THEN
       "PCS1".wMod1Flt1 := #wMF1;
       "PCS1".wMod1Flt2 := #wMF2;
       "PCS1".wMod1Flt3 := #wMF3;
       "PCS1".wMod1Flt4 := #wMF4;
   END_IF;
END_REGION

REGION Network 6: Module 2 Faults
   RUNG wire#powerrail
      { S7_Templates := "SrcType := Int" } EQ_Contact(in1 := "PCS1".iModFlt, in2 := 2)
      wire#w1
      Move(in := #wMF1, out1 => "PCS1".wMod2Flt1)
      Move(in := #wMF2, out1 => "PCS1".wMod2Flt2)
   END_RUNG
   RUNG wire#w1
      Move(in := #wMF3, out1 => "PCS1".wMod2Flt3)
      Move(in := #wMF4, out1 => "PCS1".wMod2Flt4)
   END_RUNG
   // the same network as SCL:
   IF "PCS1".iModFlt = 2 THEN
       "PCS1".wMod2Flt1 := #wMF1;
       "PCS1".wMod2Flt2 := #wMF2;
       "PCS1".wMod2Flt3 := #wMF3;
       "PCS1".wMod2Flt4 := #wMF4;
   END_IF;
END_REGION

REGION Network 7: Module 3 Faults
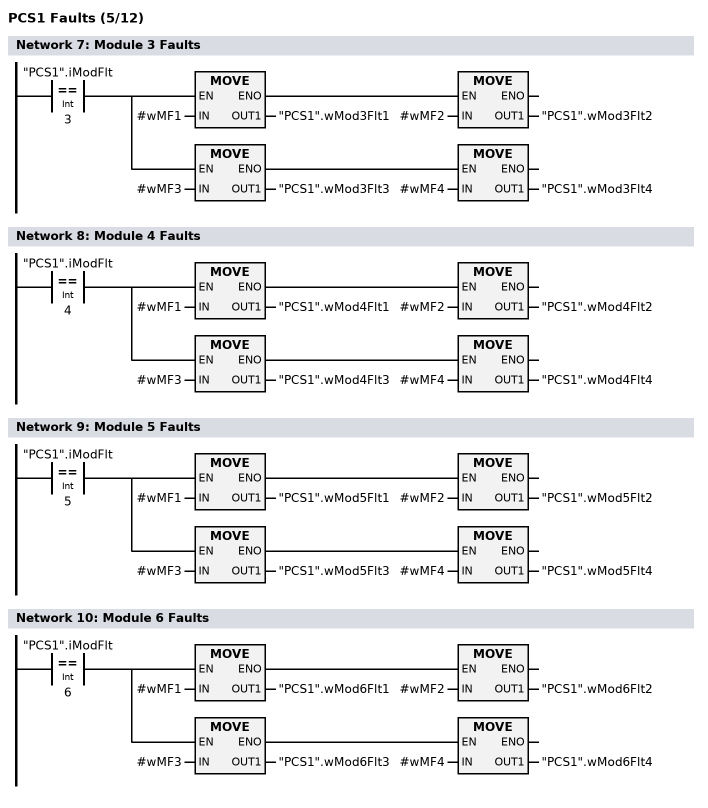
   RUNG wire#powerrail
      { S7_Templates := "SrcType := Int" } EQ_Contact(in1 := "PCS1".iModFlt, in2 := 3)
      wire#w1
      Move(in := #wMF1, out1 => "PCS1".wMod3Flt1)
      Move(in := #wMF2, out1 => "PCS1".wMod3Flt2)
   END_RUNG
   RUNG wire#w1
      Move(in := #wMF3, out1 => "PCS1".wMod3Flt3)
      Move(in := #wMF4, out1 => "PCS1".wMod3Flt4)
   END_RUNG
   // the same network as SCL:
   IF "PCS1".iModFlt = 3 THEN
       "PCS1".wMod3Flt1 := #wMF1;
       "PCS1".wMod3Flt2 := #wMF2;
       "PCS1".wMod3Flt3 := #wMF3;
       "PCS1".wMod3Flt4 := #wMF4;
   END_IF;
END_REGION

REGION Network 8: Module 4 Faults
   RUNG wire#powerrail
      { S7_Templates := "SrcType := Int" } EQ_Contact(in1 := "PCS1".iModFlt, in2 := 4)
      wire#w1
      Move(in := #wMF1, out1 => "PCS1".wMod4Flt1)
      Move(in := #wMF2, out1 => "PCS1".wMod4Flt2)
   END_RUNG
   RUNG wire#w1
      Move(in := #wMF3, out1 => "PCS1".wMod4Flt3)
      Move(in := #wMF4, out1 => "PCS1".wMod4Flt4)
   END_RUNG
   // the same network as SCL:
   IF "PCS1".iModFlt = 4 THEN
       "PCS1".wMod4Flt1 := #wMF1;
       "PCS1".wMod4Flt2 := #wMF2;
       "PCS1".wMod4Flt3 := #wMF3;
       "PCS1".wMod4Flt4 := #wMF4;
   END_IF;
END_REGION

REGION Network 9: Module 5 Faults
   RUNG wire#powerrail
      { S7_Templates := "SrcType := Int" } EQ_Contact(in1 := "PCS1".iModFlt, in2 := 5)
      wire#w1
      Move(in := #wMF1, out1 => "PCS1".wMod5Flt1)
      Move(in := #wMF2, out1 => "PCS1".wMod5Flt2)
   END_RUNG
   RUNG wire#w1
      Move(in := #wMF3, out1 => "PCS1".wMod5Flt3)
      Move(in := #wMF4, out1 => "PCS1".wMod5Flt4)
   END_RUNG
   // the same network as SCL:
   IF "PCS1".iModFlt = 5 THEN
       "PCS1".wMod5Flt1 := #wMF1;
       "PCS1".wMod5Flt2 := #wMF2;
       "PCS1".wMod5Flt3 := #wMF3;
       "PCS1".wMod5Flt4 := #wMF4;
   END_IF;
END_REGION

REGION Network 10: Module 6 Faults
   RUNG wire#powerrail
      { S7_Templates := "SrcType := Int" } EQ_Contact(in1 := "PCS1".iModFlt, in2 := 6)
      wire#w1
      Move(in := #wMF1, out1 => "PCS1".wMod6Flt1)
      Move(in := #wMF2, out1 => "PCS1".wMod6Flt2)
   END_RUNG
   RUNG wire#w1
      Move(in := #wMF3, out1 => "PCS1".wMod6Flt3)
      Move(in := #wMF4, out1 => "PCS1".wMod6Flt4)
   END_RUNG
   // the same network as SCL:
   IF "PCS1".iModFlt = 6 THEN
       "PCS1".wMod6Flt1 := #wMF1;
       "PCS1".wMod6Flt2 := #wMF2;
       "PCS1".wMod6Flt3 := #wMF3;
       "PCS1".wMod6Flt4 := #wMF4;
   END_IF;
END_REGION

REGION Network 11: Module Warnings
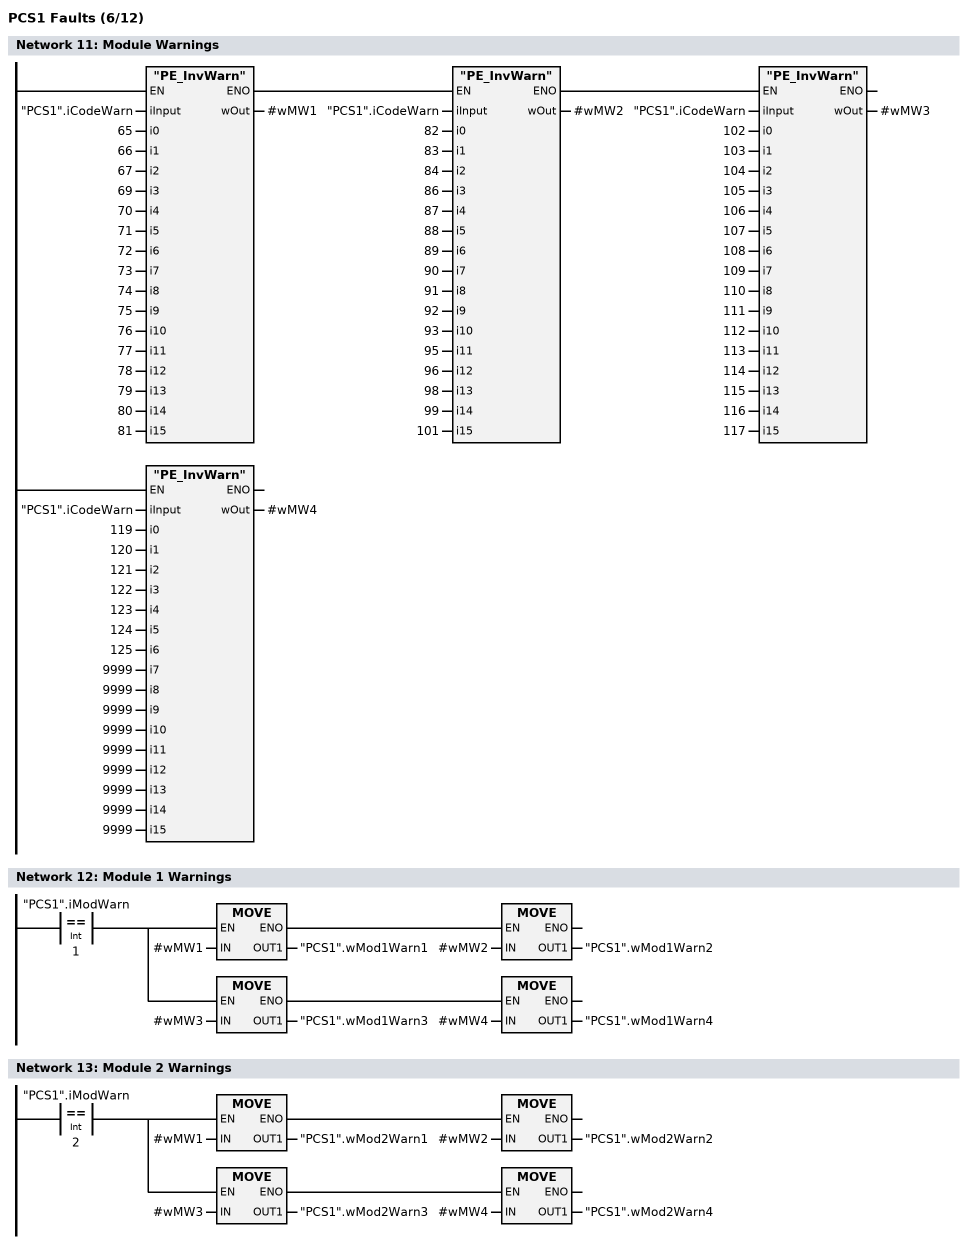
   RUNG wire#powerrail
      "PE_InvWarn"(iInput := "PCS1".iCodeWarn, i0 := 65, i1 := 66, i2 := 67, i3 := 69, i4 := 70, i5 := 71, i6 := 72, i7 := 73, i8 := 74, i9 := 75, i10 := 76, i11 := 77, i12 := 78, i13 := 79, i14 := 80, i15 := 81, wOut => #wMW1)
      "PE_InvWarn"(iInput := "PCS1".iCodeWarn, i0 := 82, i1 := 83, i2 := 84, i3 := 86, i4 := 87, i5 := 88, i6 := 89, i7 := 90, i8 := 91, i9 := 92, i10 := 93, i11 := 95, i12 := 96, i13 := 98, i14 := 99, i15 := 101, wOut => #wMW2)
      "PE_InvWarn"(iInput := "PCS1".iCodeWarn, i0 := 102, i1 := 103, i2 := 104, i3 := 105, i4 := 106, i5 := 107, i6 := 108, i7 := 109, i8 := 110, i9 := 111, i10 := 112, i11 := 113, i12 := 114, i13 := 115, i14 := 116, i15 := 117, wOut => #wMW3)
   END_RUNG
   RUNG wire#powerrail
      "PE_InvWarn"(iInput := "PCS1".iCodeWarn, i0 := 119, i1 := 120, i2 := 121, i3 := 122, i4 := 123, i5 := 124, i6 := 125, i7 := 9999, i8 := 9999, i9 := 9999, i10 := 9999, i11 := 9999, i12 := 9999, i13 := 9999, i14 := 9999, i15 := 9999, wOut => #wMW4)
   END_RUNG
   // the same network as SCL:
   "PE_InvWarn"(iInput := "PCS1".iCodeWarn,
                i0 := 65,
                i1 := 66,
                i2 := 67,
                i3 := 69,
                i4 := 70,
                i5 := 71,
                i6 := 72,
                i7 := 73,
                i8 := 74,
                i9 := 75,
                i10 := 76,
                i11 := 77,
                i12 := 78,
                i13 := 79,
                i14 := 80,
                i15 := 81,
                wOut => #wMW1,
                ENO => #_w1);
   "PE_InvWarn"(EN := #_w1,
                iInput := "PCS1".iCodeWarn,
                i0 := 82,
                i1 := 83,
                i2 := 84,
                i3 := 86,
                i4 := 87,
                i5 := 88,
                i6 := 89,
                i7 := 90,
                i8 := 91,
                i9 := 92,
                i10 := 93,
                i11 := 95,
                i12 := 96,
                i13 := 98,
                i14 := 99,
                i15 := 101,
                wOut => #wMW2,
                ENO => #_w2);
   IF #_w2 THEN
       "PE_InvWarn"(iInput := "PCS1".iCodeWarn,
                    i0 := 102,
                    i1 := 103,
                    i2 := 104,
                    i3 := 105,
                    i4 := 106,
                    i5 := 107,
                    i6 := 108,
                    i7 := 109,
                    i8 := 110,
                    i9 := 111,
                    i10 := 112,
                    i11 := 113,
                    i12 := 114,
                    i13 := 115,
                    i14 := 116,
                    i15 := 117,
                    wOut => #wMW3);
   END_IF;
   "PE_InvWarn"(iInput := "PCS1".iCodeWarn,
                i0 := 119,
                i1 := 120,
                i2 := 121,
                i3 := 122,
                i4 := 123,
                i5 := 124,
                i6 := 125,
                i7 := 9999,
                i8 := 9999,
                i9 := 9999,
                i10 := 9999,
                i11 := 9999,
                i12 := 9999,
                i13 := 9999,
                i14 := 9999,
                i15 := 9999,
                wOut => #wMW4);
END_REGION

REGION Network 12: Module 1 Warnings
   RUNG wire#powerrail
      { S7_Templates := "SrcType := Int" } EQ_Contact(in1 := "PCS1".iModWarn, in2 := 1)
      wire#w1
      Move(in := #wMW1, out1 => "PCS1".wMod1Warn1)
      Move(in := #wMW2, out1 => "PCS1".wMod1Warn2)
   END_RUNG
   RUNG wire#w1
      Move(in := #wMW3, out1 => "PCS1".wMod1Warn3)
      Move(in := #wMW4, out1 => "PCS1".wMod1Warn4)
   END_RUNG
   // the same network as SCL:
   IF "PCS1".iModWarn = 1 THEN
       "PCS1".wMod1Warn1 := #wMW1;
       "PCS1".wMod1Warn2 := #wMW2;
       "PCS1".wMod1Warn3 := #wMW3;
       "PCS1".wMod1Warn4 := #wMW4;
   END_IF;
END_REGION

REGION Network 13: Module 2 Warnings
   RUNG wire#powerrail
      { S7_Templates := "SrcType := Int" } EQ_Contact(in1 := "PCS1".iModWarn, in2 := 2)
      wire#w1
      Move(in := #wMW1, out1 => "PCS1".wMod2Warn1)
      Move(in := #wMW2, out1 => "PCS1".wMod2Warn2)
   END_RUNG
   RUNG wire#w1
      Move(in := #wMW3, out1 => "PCS1".wMod2Warn3)
      Move(in := #wMW4, out1 => "PCS1".wMod2Warn4)
   END_RUNG
   // the same network as SCL:
   IF "PCS1".iModWarn = 2 THEN
       "PCS1".wMod2Warn1 := #wMW1;
       "PCS1".wMod2Warn2 := #wMW2;
       "PCS1".wMod2Warn3 := #wMW3;
       "PCS1".wMod2Warn4 := #wMW4;
   END_IF;
END_REGION

REGION Network 14: Module 3 Warnings
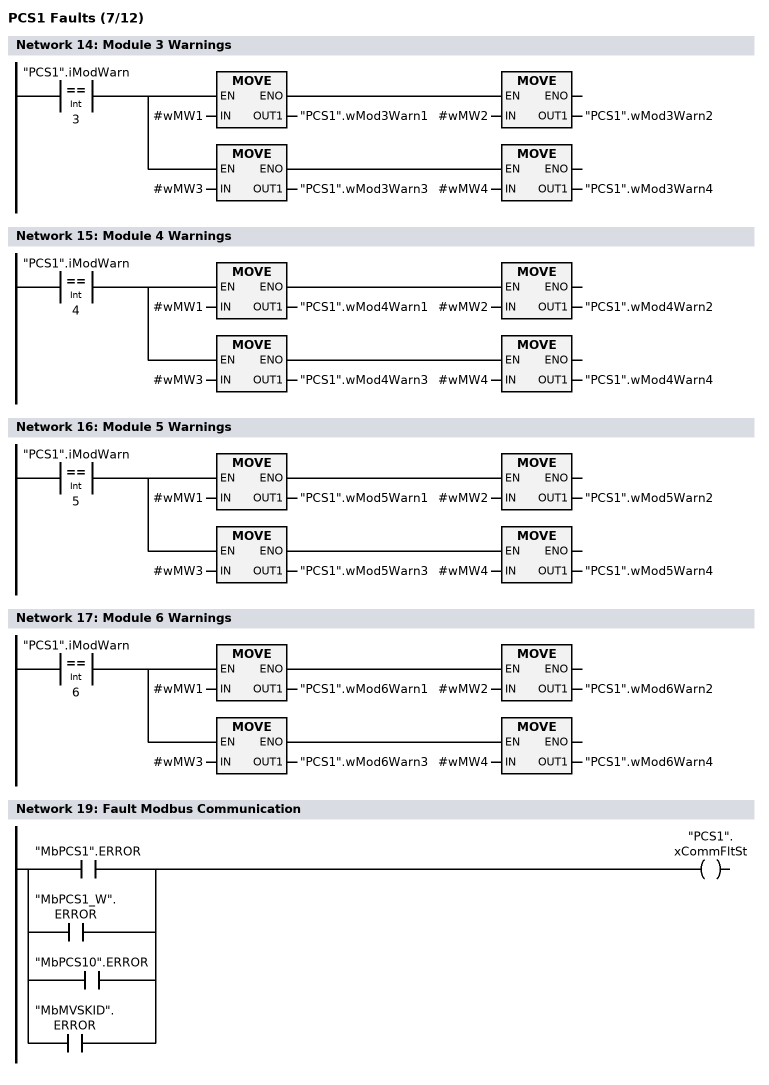
   RUNG wire#powerrail
      { S7_Templates := "SrcType := Int" } EQ_Contact(in1 := "PCS1".iModWarn, in2 := 3)
      wire#w1
      Move(in := #wMW1, out1 => "PCS1".wMod3Warn1)
      Move(in := #wMW2, out1 => "PCS1".wMod3Warn2)
   END_RUNG
   RUNG wire#w1
      Move(in := #wMW3, out1 => "PCS1".wMod3Warn3)
      Move(in := #wMW4, out1 => "PCS1".wMod3Warn4)
   END_RUNG
   // the same network as SCL:
   IF "PCS1".iModWarn = 3 THEN
       "PCS1".wMod3Warn1 := #wMW1;
       "PCS1".wMod3Warn2 := #wMW2;
       "PCS1".wMod3Warn3 := #wMW3;
       "PCS1".wMod3Warn4 := #wMW4;
   END_IF;
END_REGION

REGION Network 15: Module 4 Warnings
   RUNG wire#powerrail
      { S7_Templates := "SrcType := Int" } EQ_Contact(in1 := "PCS1".iModWarn, in2 := 4)
      wire#w1
      Move(in := #wMW1, out1 => "PCS1".wMod4Warn1)
      Move(in := #wMW2, out1 => "PCS1".wMod4Warn2)
   END_RUNG
   RUNG wire#w1
      Move(in := #wMW3, out1 => "PCS1".wMod4Warn3)
      Move(in := #wMW4, out1 => "PCS1".wMod4Warn4)
   END_RUNG
   // the same network as SCL:
   IF "PCS1".iModWarn = 4 THEN
       "PCS1".wMod4Warn1 := #wMW1;
       "PCS1".wMod4Warn2 := #wMW2;
       "PCS1".wMod4Warn3 := #wMW3;
       "PCS1".wMod4Warn4 := #wMW4;
   END_IF;
END_REGION

REGION Network 16: Module 5 Warnings
   RUNG wire#powerrail
      { S7_Templates := "SrcType := Int" } EQ_Contact(in1 := "PCS1".iModWarn, in2 := 5)
      wire#w1
      Move(in := #wMW1, out1 => "PCS1".wMod5Warn1)
      Move(in := #wMW2, out1 => "PCS1".wMod5Warn2)
   END_RUNG
   RUNG wire#w1
      Move(in := #wMW3, out1 => "PCS1".wMod5Warn3)
      Move(in := #wMW4, out1 => "PCS1".wMod5Warn4)
   END_RUNG
   // the same network as SCL:
   IF "PCS1".iModWarn = 5 THEN
       "PCS1".wMod5Warn1 := #wMW1;
       "PCS1".wMod5Warn2 := #wMW2;
       "PCS1".wMod5Warn3 := #wMW3;
       "PCS1".wMod5Warn4 := #wMW4;
   END_IF;
END_REGION

REGION Network 17: Module 6 Warnings
   RUNG wire#powerrail
      { S7_Templates := "SrcType := Int" } EQ_Contact(in1 := "PCS1".iModWarn, in2 := 6)
      wire#w1
      Move(in := #wMW1, out1 => "PCS1".wMod6Warn1)
      Move(in := #wMW2, out1 => "PCS1".wMod6Warn2)
   END_RUNG
   RUNG wire#w1
      Move(in := #wMW3, out1 => "PCS1".wMod6Warn3)
      Move(in := #wMW4, out1 => "PCS1".wMod6Warn4)
   END_RUNG
   // the same network as SCL:
   IF "PCS1".iModWarn = 6 THEN
       "PCS1".wMod6Warn1 := #wMW1;
       "PCS1".wMod6Warn2 := #wMW2;
       "PCS1".wMod6Warn3 := #wMW3;
       "PCS1".wMod6Warn4 := #wMW4;
   END_IF;
END_REGION

REGION Network 19: Fault Modbus Communication
   RUNG wire#powerrail
      Contact( "MbPCS1".ERROR )
      wire#w1
      Coil( "PCS1".xCommFltSt )
   END_RUNG
   RUNG wire#powerrail
      Contact( "MbPCS1_W".ERROR )
   END_RUNG wire#w1
   RUNG wire#powerrail
      Contact( "MbPCS10".ERROR )
   END_RUNG wire#w1
   RUNG wire#powerrail
      Contact( "MbMVSKID".ERROR )
   END_RUNG wire#w1
   // the same network as SCL:
   "PCS1".xCommFltSt := "MbPCS1".ERROR OR "MbPCS1_W".ERROR OR "MbPCS10".ERROR OR "MbMVSKID".ERROR;
END_REGION

REGION Network 20: Inverter Fault
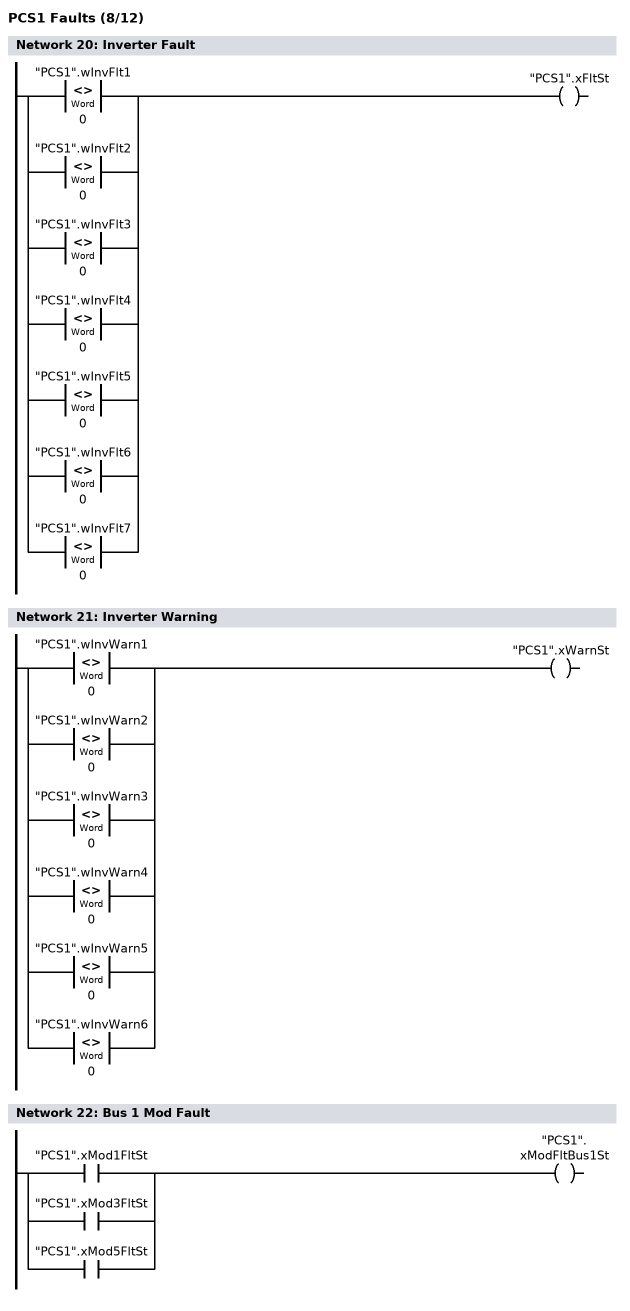
   RUNG wire#powerrail
      { S7_Templates := "SrcType := Word" } NE_Contact(in1 := "PCS1".wInvFlt1, in2 := 0)
      wire#w1
      Coil( "PCS1".xFltSt )
   END_RUNG
   RUNG wire#powerrail
      { S7_Templates := "SrcType := Word" } NE_Contact(in1 := "PCS1".wInvFlt2, in2 := 0)
   END_RUNG wire#w1
   RUNG wire#powerrail
      { S7_Templates := "SrcType := Word" } NE_Contact(in1 := "PCS1".wInvFlt3, in2 := 0)
   END_RUNG wire#w1
   RUNG wire#powerrail
      { S7_Templates := "SrcType := Word" } NE_Contact(in1 := "PCS1".wInvFlt4, in2 := 0)
   END_RUNG wire#w1
   RUNG wire#powerrail
      { S7_Templates := "SrcType := Word" } NE_Contact(in1 := "PCS1".wInvFlt5, in2 := 0)
   END_RUNG wire#w1
   RUNG wire#powerrail
      { S7_Templates := "SrcType := Word" } NE_Contact(in1 := "PCS1".wInvFlt6, in2 := 0)
   END_RUNG wire#w1
   RUNG wire#powerrail
      { S7_Templates := "SrcType := Word" } NE_Contact(in1 := "PCS1".wInvFlt7, in2 := 0)
   END_RUNG wire#w1
   // the same network as SCL:
   "PCS1".xFltSt := ("PCS1".wInvFlt1 <> 0) OR ("PCS1".wInvFlt2 <> 0) OR ("PCS1".wInvFlt3 <> 0) OR ("PCS1".wInvFlt4 <> 0) OR ("PCS1".wInvFlt5 <> 0) OR ("PCS1".wInvFlt6 <> 0) OR ("PCS1".wInvFlt7 <> 0);
END_REGION

REGION Network 21: Inverter Warning
   RUNG wire#powerrail
      { S7_Templates := "SrcType := Word" } NE_Contact(in1 := "PCS1".wInvWarn1, in2 := 0)
      wire#w1
      Coil( "PCS1".xWarnSt )
   END_RUNG
   RUNG wire#powerrail
      { S7_Templates := "SrcType := Word" } NE_Contact(in1 := "PCS1".wInvWarn2, in2 := 0)
   END_RUNG wire#w1
   RUNG wire#powerrail
      { S7_Templates := "SrcType := Word" } NE_Contact(in1 := "PCS1".wInvWarn3, in2 := 0)
   END_RUNG wire#w1
   RUNG wire#powerrail
      { S7_Templates := "SrcType := Word" } NE_Contact(in1 := "PCS1".wInvWarn4, in2 := 0)
   END_RUNG wire#w1
   RUNG wire#powerrail
      { S7_Templates := "SrcType := Word" } NE_Contact(in1 := "PCS1".wInvWarn5, in2 := 0)
   END_RUNG wire#w1
   RUNG wire#powerrail
      { S7_Templates := "SrcType := Word" } NE_Contact(in1 := "PCS1".wInvWarn6, in2 := 0)
   END_RUNG wire#w1
   // the same network as SCL:
   "PCS1".xWarnSt := ("PCS1".wInvWarn1 <> 0) OR ("PCS1".wInvWarn2 <> 0) OR ("PCS1".wInvWarn3 <> 0) OR ("PCS1".wInvWarn4 <> 0) OR ("PCS1".wInvWarn5 <> 0) OR ("PCS1".wInvWarn6 <> 0);
END_REGION

REGION Network 22: Bus 1 Mod Fault
   RUNG wire#powerrail
      Contact( "PCS1".xMod1FltSt )
      wire#w1
      Coil( "PCS1".xModFltBus1St )
   END_RUNG
   RUNG wire#powerrail
      Contact( "PCS1".xMod3FltSt )
   END_RUNG wire#w1
   RUNG wire#powerrail
      Contact( "PCS1".xMod5FltSt )
   END_RUNG wire#w1
   // the same network as SCL:
   "PCS1".xModFltBus1St := "PCS1".xMod1FltSt OR "PCS1".xMod3FltSt OR "PCS1".xMod5FltSt;
END_REGION

REGION Network 23: Bus 2 Mod Fault
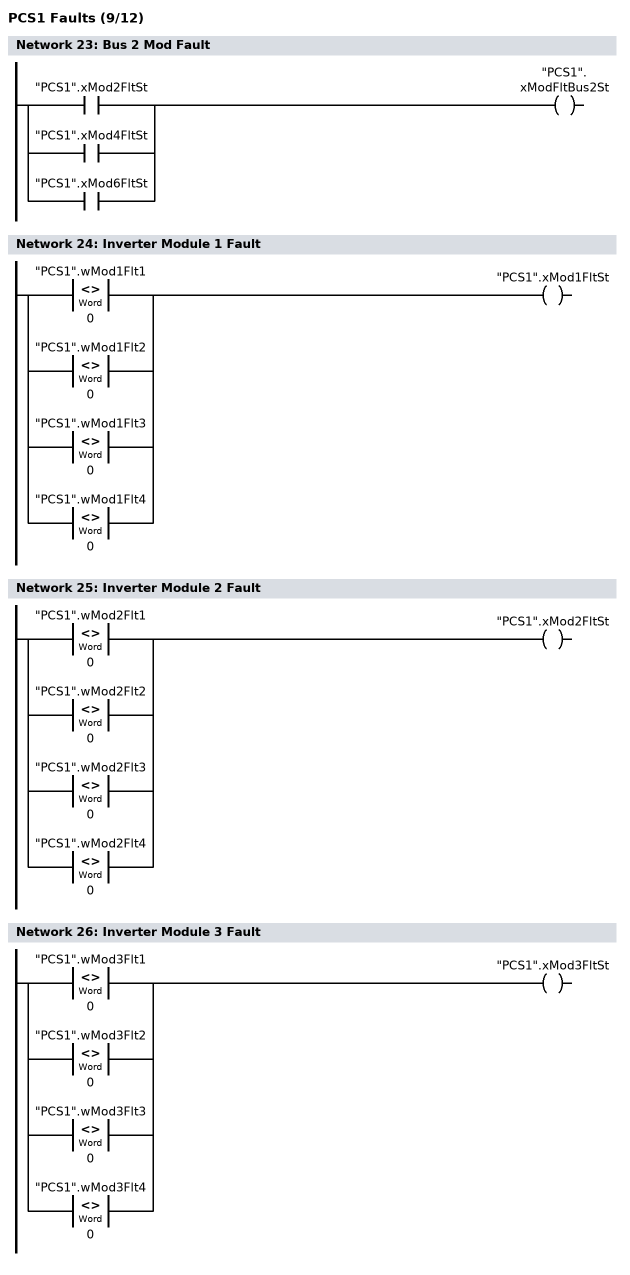
   RUNG wire#powerrail
      Contact( "PCS1".xMod2FltSt )
      wire#w1
      Coil( "PCS1".xModFltBus2St )
   END_RUNG
   RUNG wire#powerrail
      Contact( "PCS1".xMod4FltSt )
   END_RUNG wire#w1
   RUNG wire#powerrail
      Contact( "PCS1".xMod6FltSt )
   END_RUNG wire#w1
   // the same network as SCL:
   "PCS1".xModFltBus2St := "PCS1".xMod2FltSt OR "PCS1".xMod4FltSt OR "PCS1".xMod6FltSt;
END_REGION

REGION Network 24: Inverter Module 1 Fault
   RUNG wire#powerrail
      { S7_Templates := "SrcType := Word" } NE_Contact(in1 := "PCS1".wMod1Flt1, in2 := 0)
      wire#w1
      Coil( "PCS1".xMod1FltSt )
   END_RUNG
   RUNG wire#powerrail
      { S7_Templates := "SrcType := Word" } NE_Contact(in1 := "PCS1".wMod1Flt2, in2 := 0)
   END_RUNG wire#w1
   RUNG wire#powerrail
      { S7_Templates := "SrcType := Word" } NE_Contact(in1 := "PCS1".wMod1Flt3, in2 := 0)
   END_RUNG wire#w1
   RUNG wire#powerrail
      { S7_Templates := "SrcType := Word" } NE_Contact(in1 := "PCS1".wMod1Flt4, in2 := 0)
   END_RUNG wire#w1
   // the same network as SCL:
   "PCS1".xMod1FltSt := ("PCS1".wMod1Flt1 <> 0) OR ("PCS1".wMod1Flt2 <> 0) OR ("PCS1".wMod1Flt3 <> 0) OR ("PCS1".wMod1Flt4 <> 0);
END_REGION

REGION Network 25: Inverter Module 2 Fault
   RUNG wire#powerrail
      { S7_Templates := "SrcType := Word" } NE_Contact(in1 := "PCS1".wMod2Flt1, in2 := 0)
      wire#w1
      Coil( "PCS1".xMod2FltSt )
   END_RUNG
   RUNG wire#powerrail
      { S7_Templates := "SrcType := Word" } NE_Contact(in1 := "PCS1".wMod2Flt2, in2 := 0)
   END_RUNG wire#w1
   RUNG wire#powerrail
      { S7_Templates := "SrcType := Word" } NE_Contact(in1 := "PCS1".wMod2Flt3, in2 := 0)
   END_RUNG wire#w1
   RUNG wire#powerrail
      { S7_Templates := "SrcType := Word" } NE_Contact(in1 := "PCS1".wMod2Flt4, in2 := 0)
   END_RUNG wire#w1
   // the same network as SCL:
   "PCS1".xMod2FltSt := ("PCS1".wMod2Flt1 <> 0) OR ("PCS1".wMod2Flt2 <> 0) OR ("PCS1".wMod2Flt3 <> 0) OR ("PCS1".wMod2Flt4 <> 0);
END_REGION

REGION Network 26: Inverter Module 3 Fault
   RUNG wire#powerrail
      { S7_Templates := "SrcType := Word" } NE_Contact(in1 := "PCS1".wMod3Flt1, in2 := 0)
      wire#w1
      Coil( "PCS1".xMod3FltSt )
   END_RUNG
   RUNG wire#powerrail
      { S7_Templates := "SrcType := Word" } NE_Contact(in1 := "PCS1".wMod3Flt2, in2 := 0)
   END_RUNG wire#w1
   RUNG wire#powerrail
      { S7_Templates := "SrcType := Word" } NE_Contact(in1 := "PCS1".wMod3Flt3, in2 := 0)
   END_RUNG wire#w1
   RUNG wire#powerrail
      { S7_Templates := "SrcType := Word" } NE_Contact(in1 := "PCS1".wMod3Flt4, in2 := 0)
   END_RUNG wire#w1
   // the same network as SCL:
   "PCS1".xMod3FltSt := ("PCS1".wMod3Flt1 <> 0) OR ("PCS1".wMod3Flt2 <> 0) OR ("PCS1".wMod3Flt3 <> 0) OR ("PCS1".wMod3Flt4 <> 0);
END_REGION

REGION Network 27: Inverter Module 4 Fault
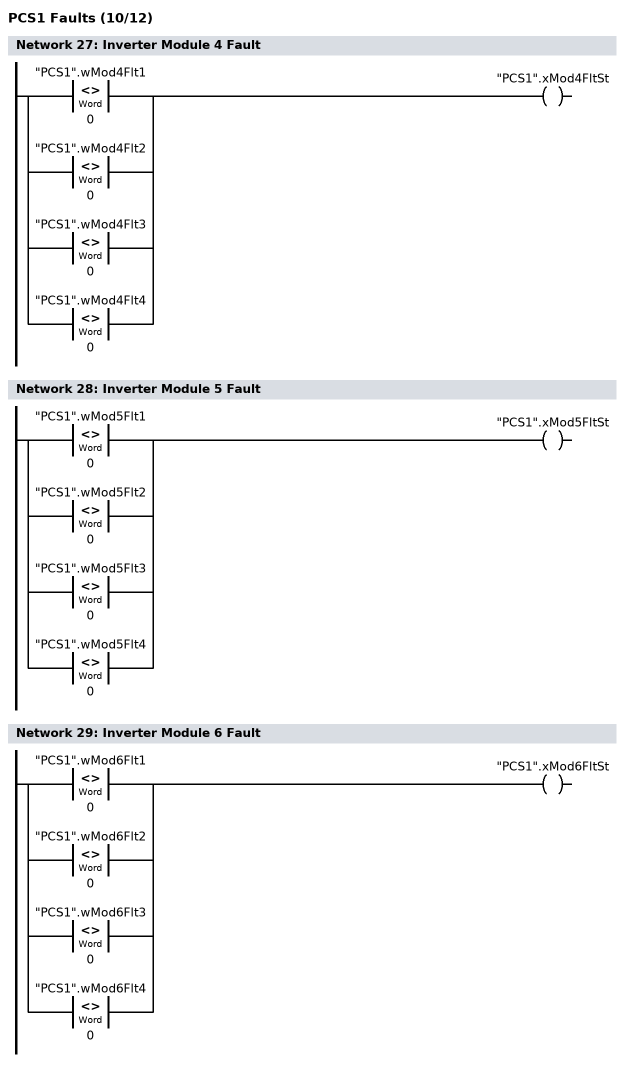
   RUNG wire#powerrail
      { S7_Templates := "SrcType := Word" } NE_Contact(in1 := "PCS1".wMod4Flt1, in2 := 0)
      wire#w1
      Coil( "PCS1".xMod4FltSt )
   END_RUNG
   RUNG wire#powerrail
      { S7_Templates := "SrcType := Word" } NE_Contact(in1 := "PCS1".wMod4Flt2, in2 := 0)
   END_RUNG wire#w1
   RUNG wire#powerrail
      { S7_Templates := "SrcType := Word" } NE_Contact(in1 := "PCS1".wMod4Flt3, in2 := 0)
   END_RUNG wire#w1
   RUNG wire#powerrail
      { S7_Templates := "SrcType := Word" } NE_Contact(in1 := "PCS1".wMod4Flt4, in2 := 0)
   END_RUNG wire#w1
   // the same network as SCL:
   "PCS1".xMod4FltSt := ("PCS1".wMod4Flt1 <> 0) OR ("PCS1".wMod4Flt2 <> 0) OR ("PCS1".wMod4Flt3 <> 0) OR ("PCS1".wMod4Flt4 <> 0);
END_REGION

REGION Network 28: Inverter Module 5 Fault
   RUNG wire#powerrail
      { S7_Templates := "SrcType := Word" } NE_Contact(in1 := "PCS1".wMod5Flt1, in2 := 0)
      wire#w1
      Coil( "PCS1".xMod5FltSt )
   END_RUNG
   RUNG wire#powerrail
      { S7_Templates := "SrcType := Word" } NE_Contact(in1 := "PCS1".wMod5Flt2, in2 := 0)
   END_RUNG wire#w1
   RUNG wire#powerrail
      { S7_Templates := "SrcType := Word" } NE_Contact(in1 := "PCS1".wMod5Flt3, in2 := 0)
   END_RUNG wire#w1
   RUNG wire#powerrail
      { S7_Templates := "SrcType := Word" } NE_Contact(in1 := "PCS1".wMod5Flt4, in2 := 0)
   END_RUNG wire#w1
   // the same network as SCL:
   "PCS1".xMod5FltSt := ("PCS1".wMod5Flt1 <> 0) OR ("PCS1".wMod5Flt2 <> 0) OR ("PCS1".wMod5Flt3 <> 0) OR ("PCS1".wMod5Flt4 <> 0);
END_REGION

REGION Network 29: Inverter Module 6 Fault
   RUNG wire#powerrail
      { S7_Templates := "SrcType := Word" } NE_Contact(in1 := "PCS1".wMod6Flt1, in2 := 0)
      wire#w1
      Coil( "PCS1".xMod6FltSt )
   END_RUNG
   RUNG wire#powerrail
      { S7_Templates := "SrcType := Word" } NE_Contact(in1 := "PCS1".wMod6Flt2, in2 := 0)
   END_RUNG wire#w1
   RUNG wire#powerrail
      { S7_Templates := "SrcType := Word" } NE_Contact(in1 := "PCS1".wMod6Flt3, in2 := 0)
   END_RUNG wire#w1
   RUNG wire#powerrail
      { S7_Templates := "SrcType := Word" } NE_Contact(in1 := "PCS1".wMod6Flt4, in2 := 0)
   END_RUNG wire#w1
   // the same network as SCL:
   "PCS1".xMod6FltSt := ("PCS1".wMod6Flt1 <> 0) OR ("PCS1".wMod6Flt2 <> 0) OR ("PCS1".wMod6Flt3 <> 0) OR ("PCS1".wMod6Flt4 <> 0);
END_REGION

REGION Network 30: Inverter Module 1 Warning
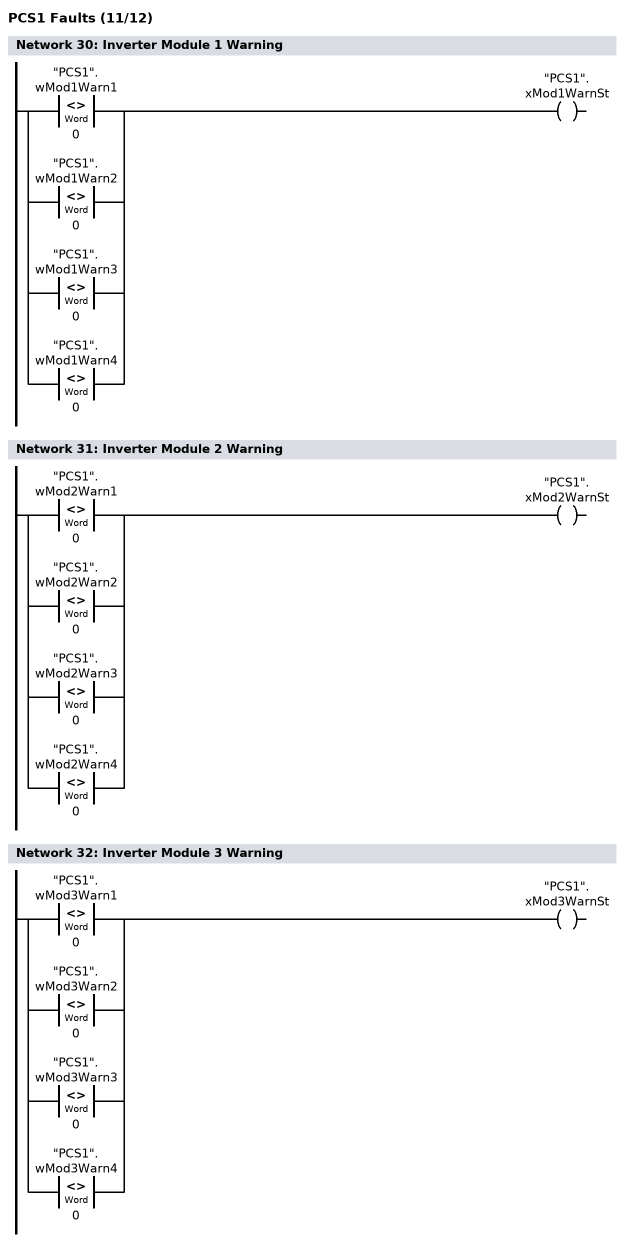
   RUNG wire#powerrail
      { S7_Templates := "SrcType := Word" } NE_Contact(in1 := "PCS1".wMod1Warn1, in2 := 0)
      wire#w1
      Coil( "PCS1".xMod1WarnSt )
   END_RUNG
   RUNG wire#powerrail
      { S7_Templates := "SrcType := Word" } NE_Contact(in1 := "PCS1".wMod1Warn2, in2 := 0)
   END_RUNG wire#w1
   RUNG wire#powerrail
      { S7_Templates := "SrcType := Word" } NE_Contact(in1 := "PCS1".wMod1Warn3, in2 := 0)
   END_RUNG wire#w1
   RUNG wire#powerrail
      { S7_Templates := "SrcType := Word" } NE_Contact(in1 := "PCS1".wMod1Warn4, in2 := 0)
   END_RUNG wire#w1
   // the same network as SCL:
   "PCS1".xMod1WarnSt := ("PCS1".wMod1Warn1 <> 0) OR ("PCS1".wMod1Warn2 <> 0) OR ("PCS1".wMod1Warn3 <> 0) OR ("PCS1".wMod1Warn4 <> 0);
END_REGION

REGION Network 31: Inverter Module 2 Warning
   RUNG wire#powerrail
      { S7_Templates := "SrcType := Word" } NE_Contact(in1 := "PCS1".wMod2Warn1, in2 := 0)
      wire#w1
      Coil( "PCS1".xMod2WarnSt )
   END_RUNG
   RUNG wire#powerrail
      { S7_Templates := "SrcType := Word" } NE_Contact(in1 := "PCS1".wMod2Warn2, in2 := 0)
   END_RUNG wire#w1
   RUNG wire#powerrail
      { S7_Templates := "SrcType := Word" } NE_Contact(in1 := "PCS1".wMod2Warn3, in2 := 0)
   END_RUNG wire#w1
   RUNG wire#powerrail
      { S7_Templates := "SrcType := Word" } NE_Contact(in1 := "PCS1".wMod2Warn4, in2 := 0)
   END_RUNG wire#w1
   // the same network as SCL:
   "PCS1".xMod2WarnSt := ("PCS1".wMod2Warn1 <> 0) OR ("PCS1".wMod2Warn2 <> 0) OR ("PCS1".wMod2Warn3 <> 0) OR ("PCS1".wMod2Warn4 <> 0);
END_REGION

REGION Network 32: Inverter Module 3 Warning
   RUNG wire#powerrail
      { S7_Templates := "SrcType := Word" } NE_Contact(in1 := "PCS1".wMod3Warn1, in2 := 0)
      wire#w1
      Coil( "PCS1".xMod3WarnSt )
   END_RUNG
   RUNG wire#powerrail
      { S7_Templates := "SrcType := Word" } NE_Contact(in1 := "PCS1".wMod3Warn2, in2 := 0)
   END_RUNG wire#w1
   RUNG wire#powerrail
      { S7_Templates := "SrcType := Word" } NE_Contact(in1 := "PCS1".wMod3Warn3, in2 := 0)
   END_RUNG wire#w1
   RUNG wire#powerrail
      { S7_Templates := "SrcType := Word" } NE_Contact(in1 := "PCS1".wMod3Warn4, in2 := 0)
   END_RUNG wire#w1
   // the same network as SCL:
   "PCS1".xMod3WarnSt := ("PCS1".wMod3Warn1 <> 0) OR ("PCS1".wMod3Warn2 <> 0) OR ("PCS1".wMod3Warn3 <> 0) OR ("PCS1".wMod3Warn4 <> 0);
END_REGION

REGION Network 33: Inverter Module 4 Warning
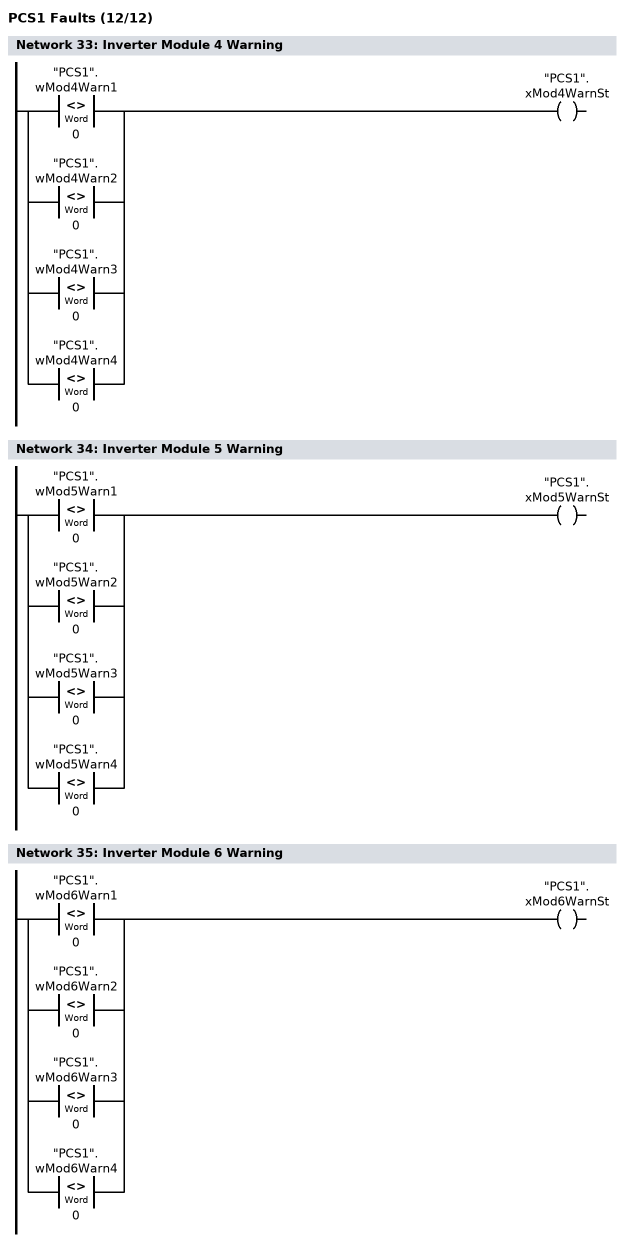
   RUNG wire#powerrail
      { S7_Templates := "SrcType := Word" } NE_Contact(in1 := "PCS1".wMod4Warn1, in2 := 0)
      wire#w1
      Coil( "PCS1".xMod4WarnSt )
   END_RUNG
   RUNG wire#powerrail
      { S7_Templates := "SrcType := Word" } NE_Contact(in1 := "PCS1".wMod4Warn2, in2 := 0)
   END_RUNG wire#w1
   RUNG wire#powerrail
      { S7_Templates := "SrcType := Word" } NE_Contact(in1 := "PCS1".wMod4Warn3, in2 := 0)
   END_RUNG wire#w1
   RUNG wire#powerrail
      { S7_Templates := "SrcType := Word" } NE_Contact(in1 := "PCS1".wMod4Warn4, in2 := 0)
   END_RUNG wire#w1
   // the same network as SCL:
   "PCS1".xMod4WarnSt := ("PCS1".wMod4Warn1 <> 0) OR ("PCS1".wMod4Warn2 <> 0) OR ("PCS1".wMod4Warn3 <> 0) OR ("PCS1".wMod4Warn4 <> 0);
END_REGION

REGION Network 34: Inverter Module 5 Warning
   RUNG wire#powerrail
      { S7_Templates := "SrcType := Word" } NE_Contact(in1 := "PCS1".wMod5Warn1, in2 := 0)
      wire#w1
      Coil( "PCS1".xMod5WarnSt )
   END_RUNG
   RUNG wire#powerrail
      { S7_Templates := "SrcType := Word" } NE_Contact(in1 := "PCS1".wMod5Warn2, in2 := 0)
   END_RUNG wire#w1
   RUNG wire#powerrail
      { S7_Templates := "SrcType := Word" } NE_Contact(in1 := "PCS1".wMod5Warn3, in2 := 0)
   END_RUNG wire#w1
   RUNG wire#powerrail
      { S7_Templates := "SrcType := Word" } NE_Contact(in1 := "PCS1".wMod5Warn4, in2 := 0)
   END_RUNG wire#w1
   // the same network as SCL:
   "PCS1".xMod5WarnSt := ("PCS1".wMod5Warn1 <> 0) OR ("PCS1".wMod5Warn2 <> 0) OR ("PCS1".wMod5Warn3 <> 0) OR ("PCS1".wMod5Warn4 <> 0);
END_REGION

REGION Network 35: Inverter Module 6 Warning
   RUNG wire#powerrail
      { S7_Templates := "SrcType := Word" } NE_Contact(in1 := "PCS1".wMod6Warn1, in2 := 0)
      wire#w1
      Coil( "PCS1".xMod6WarnSt )
   END_RUNG
   RUNG wire#powerrail
      { S7_Templates := "SrcType := Word" } NE_Contact(in1 := "PCS1".wMod6Warn2, in2 := 0)
   END_RUNG wire#w1
   RUNG wire#powerrail
      { S7_Templates := "SrcType := Word" } NE_Contact(in1 := "PCS1".wMod6Warn3, in2 := 0)
   END_RUNG wire#w1
   RUNG wire#powerrail
      { S7_Templates := "SrcType := Word" } NE_Contact(in1 := "PCS1".wMod6Warn4, in2 := 0)
   END_RUNG wire#w1
   // the same network as SCL:
   "PCS1".xMod6WarnSt := ("PCS1".wMod6Warn1 <> 0) OR ("PCS1".wMod6Warn2 <> 0) OR ("PCS1".wMod6Warn3 <> 0) OR ("PCS1".wMod6Warn4 <> 0);
END_REGION
END_FUNCTION

FUNCTION "F&Wsplit" : Void
{ S7_Optimized_Access := 'TRUE' }
VERSION : 0.1
   VAR_INPUT 
      CodeFlt : Int;
      CodeWarn : Int;
   END_VAR

   VAR_OUTPUT 
      Flt : Int;
      ModFlt : Int;
      Warn : Int;
      ModWarn : Int;
   END_VAR


BEGIN
	//Inverter Fault
	
	#Flt.%X0 := #CodeFlt.%X0;
	#Flt.%X1 := #CodeFlt.%X1;
	#Flt.%X2 := #CodeFlt.%X2;
	#Flt.%X3 := #CodeFlt.%X3;
	#Flt.%X4 := #CodeFlt.%X4;
	#Flt.%X5 := #CodeFlt.%X5;
	#Flt.%X6 := #CodeFlt.%X6;
	#Flt.%X7 := #CodeFlt.%X7;
	#Flt.%X8 := #CodeFlt.%X8;
	#Flt.%X9 := #CodeFlt.%X9;
	
	#ModFlt.%X0 := #CodeFlt.%X10;
	#ModFlt.%X1 := #CodeFlt.%X11;
	#ModFlt.%X2 := #CodeFlt.%X12;
	#ModFlt.%X3 := #CodeFlt.%X13;
	#ModFlt.%X4 := #CodeFlt.%X14;
	#ModFlt.%X5 := #CodeFlt.%X15;
	
	//Inverter Warning
	
	#Warn.%X0 := #CodeWarn.%X0;
	#Warn.%X1 := #CodeWarn.%X1;
	#Warn.%X2 := #CodeWarn.%X2;
	#Warn.%X3 := #CodeWarn.%X3;
	#Warn.%X4 := #CodeWarn.%X4;
	#Warn.%X5 := #CodeWarn.%X5;
	#Warn.%X6 := #CodeWarn.%X6;
	#Warn.%X7 := #CodeWarn.%X7;
	#Warn.%X8 := #CodeWarn.%X8;
	#Warn.%X9 := #CodeWarn.%X9;
	
	#ModWarn.%X0 := #CodeWarn.%X10;
	#ModWarn.%X1 := #CodeWarn.%X11;
	#ModWarn.%X2 := #CodeWarn.%X12;
	#ModWarn.%X3 := #CodeWarn.%X13;
	#ModWarn.%X4 := #CodeWarn.%X14;
	#ModWarn.%X5 := #CodeWarn.%X15;
	
END_FUNCTION

FUNCTION "PE_InvFlt" : Void
{ S7_Optimized_Access := 'TRUE' }
VERSION : 0.1
   VAR_INPUT 
      iInput : Int;
      i0 : Int;
      i1 : Int;
      i2 : Int;
      i3 : Int;
      i4 : Int;
      i5 : Int;
      i6 : Int;
      i7 : Int;
      i8 : Int;
      i9 : Int;
      i10 : Int;
      i11 : Int;
      i12 : Int;
      i13 : Int;
      i14 : Int;
      i15 : Int;
      xReset : Bool;
   END_VAR

   VAR_OUTPUT 
      wOut : Word;
   END_VAR


BEGIN
	
	IF #iInput = #i0
	THEN
	    #wOut.%X0 := True;
	END_IF;
	
	IF #iInput = #i1
	THEN
	    #wOut.%X1 := True;
	END_IF;
	
	IF #iInput = #i2
	THEN
	    #wOut.%X2 := True;
	END_IF;
	
	IF #iInput = #i3
	THEN
	    #wOut.%X3 := True;
	END_IF;
	
	IF #iInput = #i4
	THEN
	    #wOut.%X4 := True;
	END_IF;
	
	IF #iInput = #i5
	THEN
	    #wOut.%X5 := True;
	END_IF;
	
	IF #iInput = #i6
	THEN
	    #wOut.%X6 := True;
	END_IF;
	
	IF #iInput = #i7
	THEN
	    #wOut.%X7 := True;
	END_IF;
	
	IF #iInput = #i8
	THEN
	    #wOut.%X8 := True;
	END_IF;
	
	IF #iInput = #i9
	THEN
	    #wOut.%X9 := True;
	END_IF;
	
	IF #iInput = #i10
	THEN
	    #wOut.%X10 := True;
	END_IF;
	
	IF #iInput = #i11
	THEN
	    #wOut.%X11 := True;
	END_IF;
	
	IF #iInput = #i12
	THEN
	    #wOut.%X12 := True;
	END_IF;
	
	IF #iInput = #i13
	THEN
	    #wOut.%X13 := True;
	END_IF;
	
	IF #iInput = #i14
	THEN
	    #wOut.%X14 := True;
	END_IF;
	
	IF #iInput = #i15
	THEN
	    #wOut.%X15 := True;
	END_IF;
	
	IF #xReset
	THEN
	    #wOut := 0;
	END_IF;
	
END_FUNCTION

FUNCTION "PE_InvWarn" : Void
{ S7_Optimized_Access := 'TRUE' }
VERSION : 0.1
   VAR_INPUT 
      iInput : Int;
      i0 : Int;
      i1 : Int;
      i2 : Int;
      i3 : Int;
      i4 : Int;
      i5 : Int;
      i6 : Int;
      i7 : Int;
      i8 : Int;
      i9 : Int;
      i10 : Int;
      i11 : Int;
      i12 : Int;
      i13 : Int;
      i14 : Int;
      i15 : Int;
   END_VAR

   VAR_OUTPUT 
      wOut : Word;
   END_VAR


BEGIN
	
	#wOut.%X0 := #iInput = #i0;
	#wOut.%X1 := #iInput = #i1;
	#wOut.%X2 := #iInput = #i2;
	#wOut.%X3 := #iInput = #i3;
	#wOut.%X4 := #iInput = #i4;
	#wOut.%X5 := #iInput = #i5;
	#wOut.%X6 := #iInput = #i6;
	#wOut.%X7 := #iInput = #i7;
	#wOut.%X8 := #iInput = #i8;
	#wOut.%X9 := #iInput = #i9;
	#wOut.%X10 := #iInput = #i10;
	#wOut.%X11 := #iInput = #i11;
	#wOut.%X12 := #iInput = #i12;
	#wOut.%X13 := #iInput = #i13;
	#wOut.%X14 := #iInput = #i14;
	#wOut.%X15 := #iInput = #i15;
	
END_FUNCTION

FUNCTION "PCS1 R (PE)" : Void   // FC41, LAD
TITLE = ModBus TCP for PCS Power Electronics
{ S7_Optimized_Access := 'TRUE' }
VERSION : 0.1
// stored: AutoNumber false, IsIECCheckEnabled false, SetENOAutomatically false, UDAEnableTagReadback false
   VAR_TEMP
      rVac : Real;
   END_VAR
   VAR_TEMP   // added for the SCL form of the ladder/FBD networks
      _w1 : Bool;
   END_VAR
BEGIN

REGION Network 1: Function Modbus Client 10ms
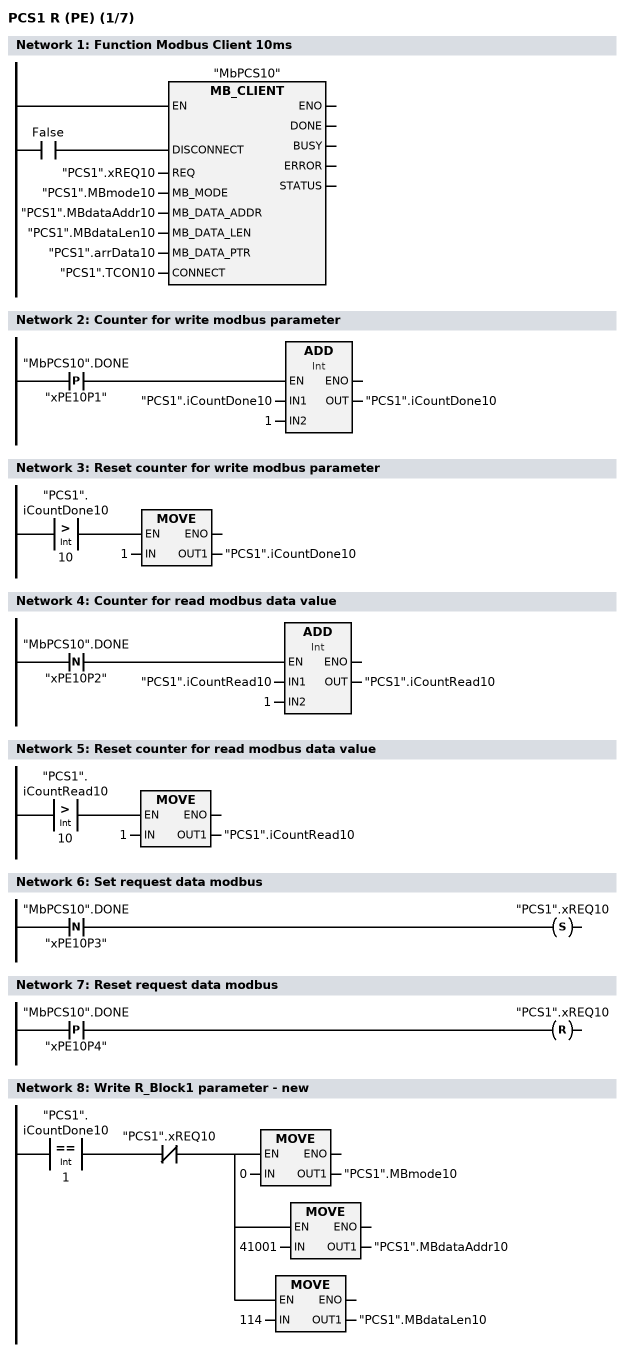
   RUNG wire#powerrail
      "MbPCS10".MB_CLIENT(DISCONNECT := wire#w1, REQ := "PCS1".xREQ10, MB_MODE := "PCS1".MBmode10, MB_DATA_ADDR := "PCS1".MBdataAddr10, MB_DATA_LEN := "PCS1".MBdataLen10, MB_DATA_PTR := "PCS1".arrData10, CONNECT := "PCS1".TCON10, DONE =>, BUSY =>, ERROR =>, STATUS =>)
   END_RUNG
   RUNG wire#powerrail
      Contact( False )
   END_RUNG wire#w1
   // the same network as SCL:
   "MbPCS10"(DISCONNECT := False,   // MB_CLIENT
             REQ := "PCS1".xREQ10,
             MB_MODE := "PCS1".MBmode10,
             MB_DATA_ADDR := "PCS1".MBdataAddr10,
             MB_DATA_LEN := "PCS1".MBdataLen10,
             MB_DATA_PTR := "PCS1".arrData10,
             CONNECT := "PCS1".TCON10);
END_REGION

REGION Network 2: Counter for write modbus parameter
   RUNG wire#powerrail
      P_Contact(operand := "MbPCS10".DONE, bit := "xPE10P1")
      { S7_Templates := "SrcType := Int" } Add(in1 := "PCS1".iCountDone10, in2 := 1, out => "PCS1".iCountDone10)
   END_RUNG
   // the same network as SCL:
   #_w1 := "MbPCS10".DONE AND NOT "xPE10P1";   // rising edge of "MbPCS10".DONE
   "xPE10P1" := "MbPCS10".DONE;
   IF #_w1 THEN "PCS1".iCountDone10 := "PCS1".iCountDone10 + 1; END_IF;
END_REGION

REGION Network 3: Reset counter for write modbus parameter
   RUNG wire#powerrail
      { S7_Templates := "SrcType := Int" } GT_Contact(in1 := "PCS1".iCountDone10, in2 := 10)
      Move(in := 1, out1 => "PCS1".iCountDone10)
   END_RUNG
   // the same network as SCL:
   IF "PCS1".iCountDone10 > 10 THEN "PCS1".iCountDone10 := 1; END_IF;
END_REGION

REGION Network 4: Counter for read modbus data value
   RUNG wire#powerrail
      N_Contact(operand := "MbPCS10".DONE, bit := "xPE10P2")
      { S7_Templates := "SrcType := Int" } Add(in1 := "PCS1".iCountRead10, in2 := 1, out => "PCS1".iCountRead10)
   END_RUNG
   // the same network as SCL:
   #_w1 := NOT "MbPCS10".DONE AND "xPE10P2";   // falling edge of "MbPCS10".DONE
   "xPE10P2" := "MbPCS10".DONE;
   IF #_w1 THEN "PCS1".iCountRead10 := "PCS1".iCountRead10 + 1; END_IF;
END_REGION

REGION Network 5: Reset counter for read modbus data value
   RUNG wire#powerrail
      { S7_Templates := "SrcType := Int" } GT_Contact(in1 := "PCS1".iCountRead10, in2 := 10)
      Move(in := 1, out1 => "PCS1".iCountRead10)
   END_RUNG
   // the same network as SCL:
   IF "PCS1".iCountRead10 > 10 THEN "PCS1".iCountRead10 := 1; END_IF;
END_REGION

REGION Network 6: Set request data modbus
   RUNG wire#powerrail
      N_Contact(operand := "MbPCS10".DONE, bit := "xPE10P3")
      S_Coil( "PCS1".xREQ10 )
   END_RUNG
   // the same network as SCL:
   #_w1 := NOT "MbPCS10".DONE AND "xPE10P3";   // falling edge of "MbPCS10".DONE
   "xPE10P3" := "MbPCS10".DONE;
   IF #_w1 THEN "PCS1".xREQ10 := TRUE; END_IF;
END_REGION

REGION Network 7: Reset request data modbus
   RUNG wire#powerrail
      P_Contact(operand := "MbPCS10".DONE, bit := "xPE10P4")
      R_Coil( "PCS1".xREQ10 )
   END_RUNG
   // the same network as SCL:
   #_w1 := "MbPCS10".DONE AND NOT "xPE10P4";   // rising edge of "MbPCS10".DONE
   "xPE10P4" := "MbPCS10".DONE;
   IF #_w1 THEN "PCS1".xREQ10 := FALSE; END_IF;
END_REGION

REGION Network 8: Write R_Block1 parameter - new
   RUNG wire#powerrail
      { S7_Templates := "SrcType := Int" } EQ_Contact(in1 := "PCS1".iCountDone10, in2 := 1)
      I_Contact( "PCS1".xREQ10 )
      wire#w1
      Move(in := 0, out1 => "PCS1".MBmode10)
   END_RUNG
   RUNG wire#w1
      Move(in := 41001, out1 => "PCS1".MBdataAddr10)
   END_RUNG
   RUNG wire#w1
      Move(in := 114, out1 => "PCS1".MBdataLen10)
   END_RUNG
   // the same network as SCL:
   IF ("PCS1".iCountDone10 = 1) AND NOT "PCS1".xREQ10 THEN
       "PCS1".MBmode10 := 0;
       "PCS1".MBdataAddr10 := 41001;
       "PCS1".MBdataLen10 := 114;
   END_IF;
END_REGION

REGION Network 9: Read R_Block1 data value - new
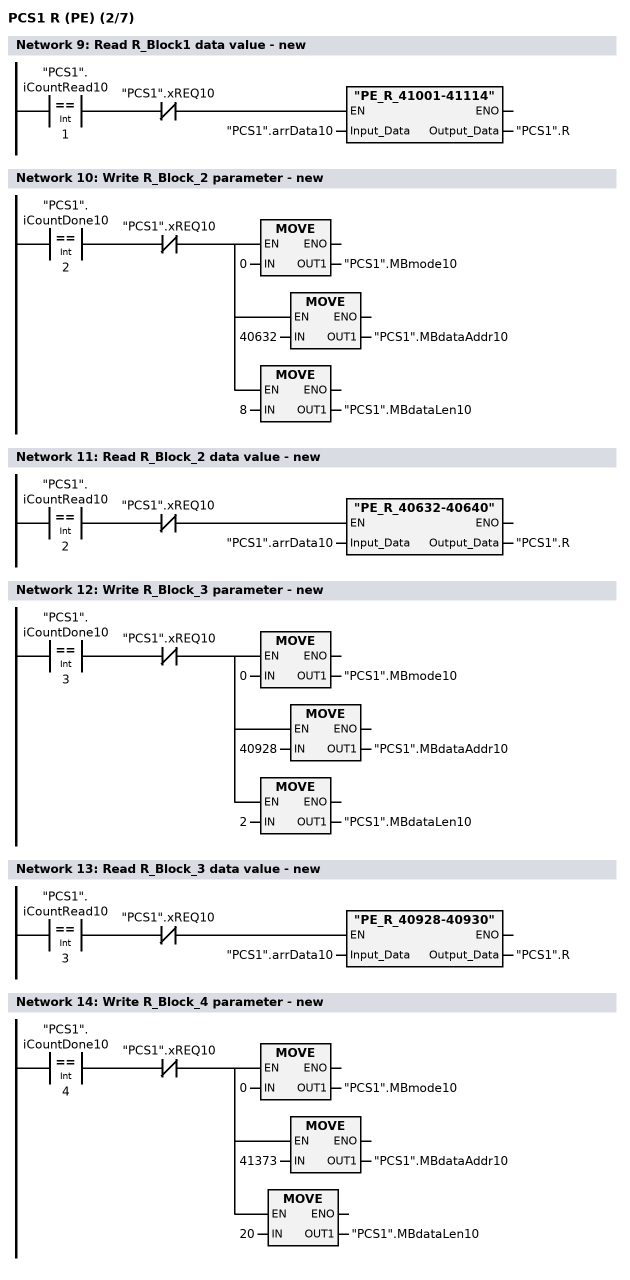
   RUNG wire#powerrail
      { S7_Templates := "SrcType := Int" } EQ_Contact(in1 := "PCS1".iCountRead10, in2 := 1)
      I_Contact( "PCS1".xREQ10 )
      "PE_R_41001-41114"(Input_Data := "PCS1".arrData10, Output_Data => "PCS1".R)
   END_RUNG
   // the same network as SCL:
   IF ("PCS1".iCountRead10 = 1) AND NOT "PCS1".xREQ10 THEN
       "PE_R_41001-41114"(Input_Data := "PCS1".arrData10, Output_Data => "PCS1".R);
   END_IF;
END_REGION

REGION Network 10: Write R_Block_2 parameter - new
   RUNG wire#powerrail
      { S7_Templates := "SrcType := Int" } EQ_Contact(in1 := "PCS1".iCountDone10, in2 := 2)
      I_Contact( "PCS1".xREQ10 )
      wire#w1
      Move(in := 0, out1 => "PCS1".MBmode10)
   END_RUNG
   RUNG wire#w1
      Move(in := 40632, out1 => "PCS1".MBdataAddr10)
   END_RUNG
   RUNG wire#w1
      Move(in := 8, out1 => "PCS1".MBdataLen10)
   END_RUNG
   // the same network as SCL:
   IF ("PCS1".iCountDone10 = 2) AND NOT "PCS1".xREQ10 THEN
       "PCS1".MBmode10 := 0;
       "PCS1".MBdataAddr10 := 40632;
       "PCS1".MBdataLen10 := 8;
   END_IF;
END_REGION

REGION Network 11: Read R_Block_2 data value - new
   RUNG wire#powerrail
      { S7_Templates := "SrcType := Int" } EQ_Contact(in1 := "PCS1".iCountRead10, in2 := 2)
      I_Contact( "PCS1".xREQ10 )
      "PE_R_40632-40640"(Input_Data := "PCS1".arrData10, Output_Data => "PCS1".R)
   END_RUNG
   // the same network as SCL:
   IF ("PCS1".iCountRead10 = 2) AND NOT "PCS1".xREQ10 THEN
       "PE_R_40632-40640"(Input_Data := "PCS1".arrData10, Output_Data => "PCS1".R);
   END_IF;
END_REGION

REGION Network 12: Write R_Block_3 parameter - new
   RUNG wire#powerrail
      { S7_Templates := "SrcType := Int" } EQ_Contact(in1 := "PCS1".iCountDone10, in2 := 3)
      I_Contact( "PCS1".xREQ10 )
      wire#w1
      Move(in := 0, out1 => "PCS1".MBmode10)
   END_RUNG
   RUNG wire#w1
      Move(in := 40928, out1 => "PCS1".MBdataAddr10)
   END_RUNG
   RUNG wire#w1
      Move(in := 2, out1 => "PCS1".MBdataLen10)
   END_RUNG
   // the same network as SCL:
   IF ("PCS1".iCountDone10 = 3) AND NOT "PCS1".xREQ10 THEN
       "PCS1".MBmode10 := 0;
       "PCS1".MBdataAddr10 := 40928;
       "PCS1".MBdataLen10 := 2;
   END_IF;
END_REGION

REGION Network 13: Read R_Block_3 data value - new
   RUNG wire#powerrail
      { S7_Templates := "SrcType := Int" } EQ_Contact(in1 := "PCS1".iCountRead10, in2 := 3)
      I_Contact( "PCS1".xREQ10 )
      "PE_R_40928-40930"(Input_Data := "PCS1".arrData10, Output_Data => "PCS1".R)
   END_RUNG
   // the same network as SCL:
   IF ("PCS1".iCountRead10 = 3) AND NOT "PCS1".xREQ10 THEN
       "PE_R_40928-40930"(Input_Data := "PCS1".arrData10, Output_Data => "PCS1".R);
   END_IF;
END_REGION

REGION Network 14: Write R_Block_4 parameter - new
   RUNG wire#powerrail
      { S7_Templates := "SrcType := Int" } EQ_Contact(in1 := "PCS1".iCountDone10, in2 := 4)
      I_Contact( "PCS1".xREQ10 )
      wire#w1
      Move(in := 0, out1 => "PCS1".MBmode10)
   END_RUNG
   RUNG wire#w1
      Move(in := 41373, out1 => "PCS1".MBdataAddr10)
   END_RUNG
   RUNG wire#w1
      Move(in := 20, out1 => "PCS1".MBdataLen10)
   END_RUNG
   // the same network as SCL:
   IF ("PCS1".iCountDone10 = 4) AND NOT "PCS1".xREQ10 THEN
       "PCS1".MBmode10 := 0;
       "PCS1".MBdataAddr10 := 41373;
       "PCS1".MBdataLen10 := 20;
   END_IF;
END_REGION

REGION Network 15: Read R_Block_4 data value - new
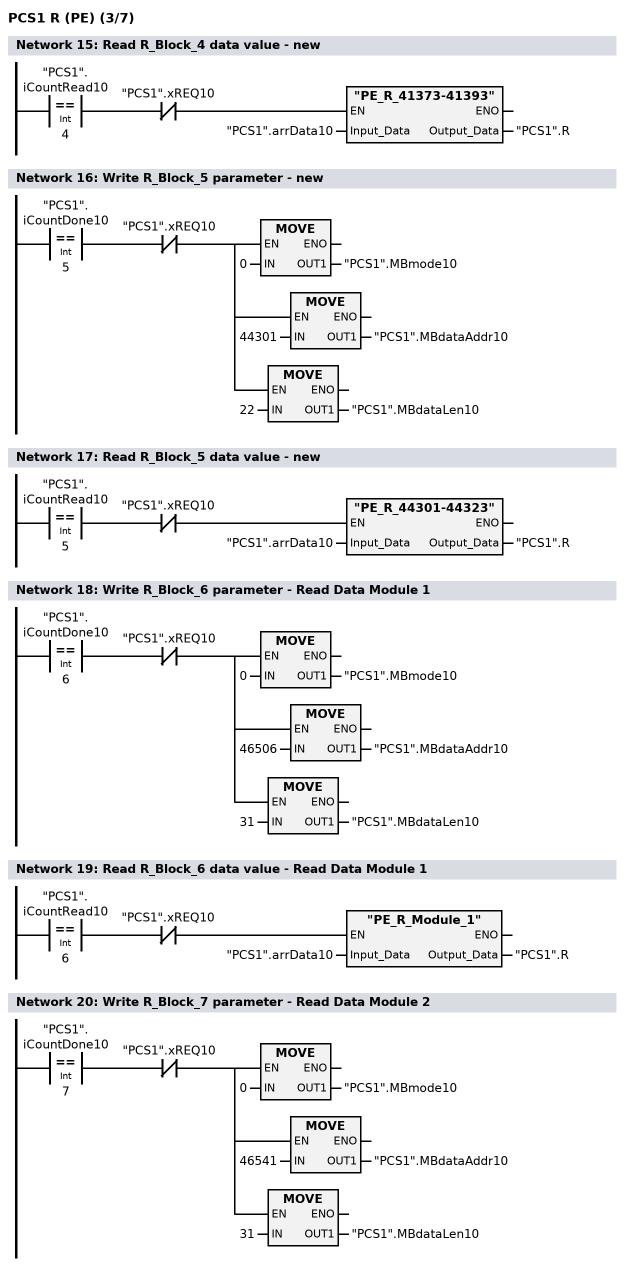
   RUNG wire#powerrail
      { S7_Templates := "SrcType := Int" } EQ_Contact(in1 := "PCS1".iCountRead10, in2 := 4)
      I_Contact( "PCS1".xREQ10 )
      "PE_R_41373-41393"(Input_Data := "PCS1".arrData10, Output_Data => "PCS1".R)
   END_RUNG
   // the same network as SCL:
   IF ("PCS1".iCountRead10 = 4) AND NOT "PCS1".xREQ10 THEN
       "PE_R_41373-41393"(Input_Data := "PCS1".arrData10, Output_Data => "PCS1".R);
   END_IF;
END_REGION

REGION Network 16: Write R_Block_5 parameter - new
   RUNG wire#powerrail
      { S7_Templates := "SrcType := Int" } EQ_Contact(in1 := "PCS1".iCountDone10, in2 := 5)
      I_Contact( "PCS1".xREQ10 )
      wire#w1
      Move(in := 0, out1 => "PCS1".MBmode10)
   END_RUNG
   RUNG wire#w1
      Move(in := 44301, out1 => "PCS1".MBdataAddr10)
   END_RUNG
   RUNG wire#w1
      Move(in := 22, out1 => "PCS1".MBdataLen10)
   END_RUNG
   // the same network as SCL:
   IF ("PCS1".iCountDone10 = 5) AND NOT "PCS1".xREQ10 THEN
       "PCS1".MBmode10 := 0;
       "PCS1".MBdataAddr10 := 44301;
       "PCS1".MBdataLen10 := 22;
   END_IF;
END_REGION

REGION Network 17: Read R_Block_5 data value - new
   RUNG wire#powerrail
      { S7_Templates := "SrcType := Int" } EQ_Contact(in1 := "PCS1".iCountRead10, in2 := 5)
      I_Contact( "PCS1".xREQ10 )
      "PE_R_44301-44323"(Input_Data := "PCS1".arrData10, Output_Data => "PCS1".R)
   END_RUNG
   // the same network as SCL:
   IF ("PCS1".iCountRead10 = 5) AND NOT "PCS1".xREQ10 THEN
       "PE_R_44301-44323"(Input_Data := "PCS1".arrData10, Output_Data => "PCS1".R);
   END_IF;
END_REGION

REGION Network 18: Write R_Block_6 parameter - Read Data Module 1
   RUNG wire#powerrail
      { S7_Templates := "SrcType := Int" } EQ_Contact(in1 := "PCS1".iCountDone10, in2 := 6)
      I_Contact( "PCS1".xREQ10 )
      wire#w1
      Move(in := 0, out1 => "PCS1".MBmode10)
   END_RUNG
   RUNG wire#w1
      Move(in := 46506, out1 => "PCS1".MBdataAddr10)
   END_RUNG
   RUNG wire#w1
      Move(in := 31, out1 => "PCS1".MBdataLen10)
   END_RUNG
   // the same network as SCL:
   IF ("PCS1".iCountDone10 = 6) AND NOT "PCS1".xREQ10 THEN
       "PCS1".MBmode10 := 0;
       "PCS1".MBdataAddr10 := 46506;
       "PCS1".MBdataLen10 := 31;
   END_IF;
END_REGION

REGION Network 19: Read R_Block_6 data value - Read Data Module 1
   RUNG wire#powerrail
      { S7_Templates := "SrcType := Int" } EQ_Contact(in1 := "PCS1".iCountRead10, in2 := 6)
      I_Contact( "PCS1".xREQ10 )
      "PE_R_Module_1"(Input_Data := "PCS1".arrData10, Output_Data => "PCS1".R)
   END_RUNG
   // the same network as SCL:
   IF ("PCS1".iCountRead10 = 6) AND NOT "PCS1".xREQ10 THEN
       "PE_R_Module_1"(Input_Data := "PCS1".arrData10, Output_Data => "PCS1".R);
   END_IF;
END_REGION

REGION Network 20: Write R_Block_7 parameter - Read Data Module 2
   RUNG wire#powerrail
      { S7_Templates := "SrcType := Int" } EQ_Contact(in1 := "PCS1".iCountDone10, in2 := 7)
      I_Contact( "PCS1".xREQ10 )
      wire#w1
      Move(in := 0, out1 => "PCS1".MBmode10)
   END_RUNG
   RUNG wire#w1
      Move(in := 46541, out1 => "PCS1".MBdataAddr10)
   END_RUNG
   RUNG wire#w1
      Move(in := 31, out1 => "PCS1".MBdataLen10)
   END_RUNG
   // the same network as SCL:
   IF ("PCS1".iCountDone10 = 7) AND NOT "PCS1".xREQ10 THEN
       "PCS1".MBmode10 := 0;
       "PCS1".MBdataAddr10 := 46541;
       "PCS1".MBdataLen10 := 31;
   END_IF;
END_REGION

REGION Network 21: Read R_Block_7 data value - Read Data Module 2
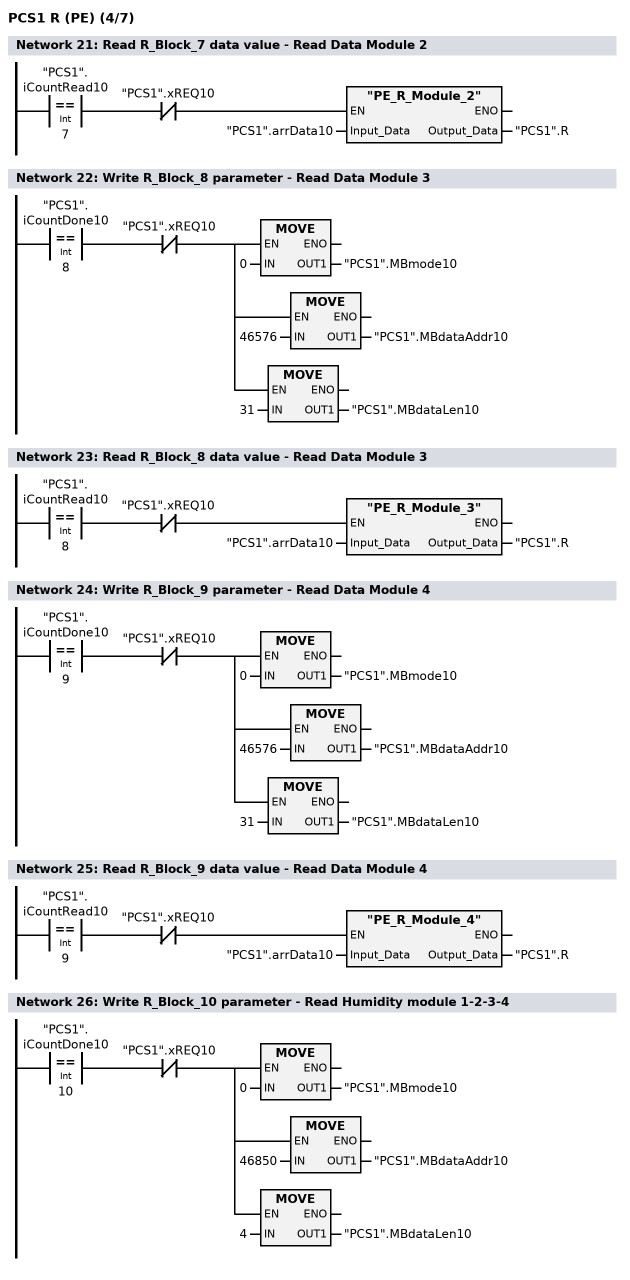
   RUNG wire#powerrail
      { S7_Templates := "SrcType := Int" } EQ_Contact(in1 := "PCS1".iCountRead10, in2 := 7)
      I_Contact( "PCS1".xREQ10 )
      "PE_R_Module_2"(Input_Data := "PCS1".arrData10, Output_Data => "PCS1".R)
   END_RUNG
   // the same network as SCL:
   IF ("PCS1".iCountRead10 = 7) AND NOT "PCS1".xREQ10 THEN
       "PE_R_Module_2"(Input_Data := "PCS1".arrData10, Output_Data => "PCS1".R);
   END_IF;
END_REGION

REGION Network 22: Write R_Block_8 parameter - Read Data Module 3
   RUNG wire#powerrail
      { S7_Templates := "SrcType := Int" } EQ_Contact(in1 := "PCS1".iCountDone10, in2 := 8)
      I_Contact( "PCS1".xREQ10 )
      wire#w1
      Move(in := 0, out1 => "PCS1".MBmode10)
   END_RUNG
   RUNG wire#w1
      Move(in := 46576, out1 => "PCS1".MBdataAddr10)
   END_RUNG
   RUNG wire#w1
      Move(in := 31, out1 => "PCS1".MBdataLen10)
   END_RUNG
   // the same network as SCL:
   IF ("PCS1".iCountDone10 = 8) AND NOT "PCS1".xREQ10 THEN
       "PCS1".MBmode10 := 0;
       "PCS1".MBdataAddr10 := 46576;
       "PCS1".MBdataLen10 := 31;
   END_IF;
END_REGION

REGION Network 23: Read R_Block_8 data value - Read Data Module 3
   RUNG wire#powerrail
      { S7_Templates := "SrcType := Int" } EQ_Contact(in1 := "PCS1".iCountRead10, in2 := 8)
      I_Contact( "PCS1".xREQ10 )
      "PE_R_Module_3"(Input_Data := "PCS1".arrData10, Output_Data => "PCS1".R)
   END_RUNG
   // the same network as SCL:
   IF ("PCS1".iCountRead10 = 8) AND NOT "PCS1".xREQ10 THEN
       "PE_R_Module_3"(Input_Data := "PCS1".arrData10, Output_Data => "PCS1".R);
   END_IF;
END_REGION

REGION Network 24: Write R_Block_9 parameter - Read Data Module 4
   RUNG wire#powerrail
      { S7_Templates := "SrcType := Int" } EQ_Contact(in1 := "PCS1".iCountDone10, in2 := 9)
      I_Contact( "PCS1".xREQ10 )
      wire#w1
      Move(in := 0, out1 => "PCS1".MBmode10)
   END_RUNG
   RUNG wire#w1
      Move(in := 46576, out1 => "PCS1".MBdataAddr10)
   END_RUNG
   RUNG wire#w1
      Move(in := 31, out1 => "PCS1".MBdataLen10)
   END_RUNG
   // the same network as SCL:
   IF ("PCS1".iCountDone10 = 9) AND NOT "PCS1".xREQ10 THEN
       "PCS1".MBmode10 := 0;
       "PCS1".MBdataAddr10 := 46576;
       "PCS1".MBdataLen10 := 31;
   END_IF;
END_REGION

REGION Network 25: Read R_Block_9 data value - Read Data Module 4
   RUNG wire#powerrail
      { S7_Templates := "SrcType := Int" } EQ_Contact(in1 := "PCS1".iCountRead10, in2 := 9)
      I_Contact( "PCS1".xREQ10 )
      "PE_R_Module_4"(Input_Data := "PCS1".arrData10, Output_Data => "PCS1".R)
   END_RUNG
   // the same network as SCL:
   IF ("PCS1".iCountRead10 = 9) AND NOT "PCS1".xREQ10 THEN
       "PE_R_Module_4"(Input_Data := "PCS1".arrData10, Output_Data => "PCS1".R);
   END_IF;
END_REGION

REGION Network 26: Write R_Block_10 parameter - Read Humidity module 1-2-3-4
   RUNG wire#powerrail
      { S7_Templates := "SrcType := Int" } EQ_Contact(in1 := "PCS1".iCountDone10, in2 := 10)
      I_Contact( "PCS1".xREQ10 )
      wire#w1
      Move(in := 0, out1 => "PCS1".MBmode10)
   END_RUNG
   RUNG wire#w1
      Move(in := 46850, out1 => "PCS1".MBdataAddr10)
   END_RUNG
   RUNG wire#w1
      Move(in := 4, out1 => "PCS1".MBdataLen10)
   END_RUNG
   // the same network as SCL:
   IF ("PCS1".iCountDone10 = 10) AND NOT "PCS1".xREQ10 THEN
       "PCS1".MBmode10 := 0;
       "PCS1".MBdataAddr10 := 46850;
       "PCS1".MBdataLen10 := 4;
   END_IF;
END_REGION

REGION Network 27: Read R_Block_10 data value - Read Humidity module 1-2-3-4
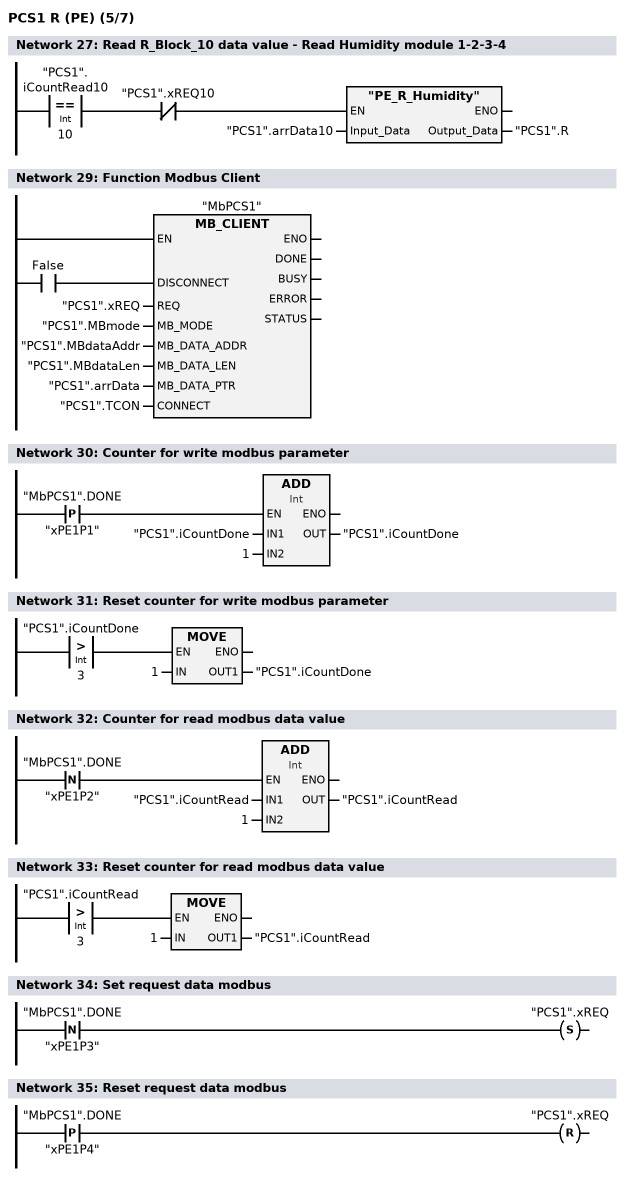
   RUNG wire#powerrail
      { S7_Templates := "SrcType := Int" } EQ_Contact(in1 := "PCS1".iCountRead10, in2 := 10)
      I_Contact( "PCS1".xREQ10 )
      "PE_R_Humidity"(Input_Data := "PCS1".arrData10, Output_Data => "PCS1".R)
   END_RUNG
   // the same network as SCL:
   IF ("PCS1".iCountRead10 = 10) AND NOT "PCS1".xREQ10 THEN
       "PE_R_Humidity"(Input_Data := "PCS1".arrData10, Output_Data => "PCS1".R);
   END_IF;
END_REGION

REGION Network 29: Function Modbus Client
   RUNG wire#powerrail
      "MbPCS1".MB_CLIENT(DISCONNECT := wire#w1, REQ := "PCS1".xREQ, MB_MODE := "PCS1".MBmode, MB_DATA_ADDR := "PCS1".MBdataAddr, MB_DATA_LEN := "PCS1".MBdataLen, MB_DATA_PTR := "PCS1".arrData, CONNECT := "PCS1".TCON, DONE =>, BUSY =>, ERROR =>, STATUS =>)
   END_RUNG
   RUNG wire#powerrail
      Contact( False )
   END_RUNG wire#w1
   // the same network as SCL:
   "MbPCS1"(DISCONNECT := False,   // MB_CLIENT
            REQ := "PCS1".xREQ,
            MB_MODE := "PCS1".MBmode,
            MB_DATA_ADDR := "PCS1".MBdataAddr,
            MB_DATA_LEN := "PCS1".MBdataLen,
            MB_DATA_PTR := "PCS1".arrData,
            CONNECT := "PCS1".TCON);
END_REGION

REGION Network 30: Counter for write modbus parameter
   RUNG wire#powerrail
      P_Contact(operand := "MbPCS1".DONE, bit := "xPE1P1")
      { S7_Templates := "SrcType := Int" } Add(in1 := "PCS1".iCountDone, in2 := 1, out => "PCS1".iCountDone)
   END_RUNG
   // the same network as SCL:
   #_w1 := "MbPCS1".DONE AND NOT "xPE1P1";   // rising edge of "MbPCS1".DONE
   "xPE1P1" := "MbPCS1".DONE;
   IF #_w1 THEN "PCS1".iCountDone := "PCS1".iCountDone + 1; END_IF;
END_REGION

REGION Network 31: Reset counter for write modbus parameter
   RUNG wire#powerrail
      { S7_Templates := "SrcType := Int" } GT_Contact(in1 := "PCS1".iCountDone, in2 := 3)
      Move(in := 1, out1 => "PCS1".iCountDone)
   END_RUNG
   // the same network as SCL:
   IF "PCS1".iCountDone > 3 THEN "PCS1".iCountDone := 1; END_IF;
END_REGION

REGION Network 32: Counter for read modbus data value
   RUNG wire#powerrail
      N_Contact(operand := "MbPCS1".DONE, bit := "xPE1P2")
      { S7_Templates := "SrcType := Int" } Add(in1 := "PCS1".iCountRead, in2 := 1, out => "PCS1".iCountRead)
   END_RUNG
   // the same network as SCL:
   #_w1 := NOT "MbPCS1".DONE AND "xPE1P2";   // falling edge of "MbPCS1".DONE
   "xPE1P2" := "MbPCS1".DONE;
   IF #_w1 THEN "PCS1".iCountRead := "PCS1".iCountRead + 1; END_IF;
END_REGION

REGION Network 33: Reset counter for read modbus data value
   RUNG wire#powerrail
      { S7_Templates := "SrcType := Int" } GT_Contact(in1 := "PCS1".iCountRead, in2 := 3)
      Move(in := 1, out1 => "PCS1".iCountRead)
   END_RUNG
   // the same network as SCL:
   IF "PCS1".iCountRead > 3 THEN "PCS1".iCountRead := 1; END_IF;
END_REGION

REGION Network 34: Set request data modbus
   RUNG wire#powerrail
      N_Contact(operand := "MbPCS1".DONE, bit := "xPE1P3")
      S_Coil( "PCS1".xREQ )
   END_RUNG
   // the same network as SCL:
   #_w1 := NOT "MbPCS1".DONE AND "xPE1P3";   // falling edge of "MbPCS1".DONE
   "xPE1P3" := "MbPCS1".DONE;
   IF #_w1 THEN "PCS1".xREQ := TRUE; END_IF;
END_REGION

REGION Network 35: Reset request data modbus
   RUNG wire#powerrail
      P_Contact(operand := "MbPCS1".DONE, bit := "xPE1P4")
      R_Coil( "PCS1".xREQ )
   END_RUNG
   // the same network as SCL:
   #_w1 := "MbPCS1".DONE AND NOT "xPE1P4";   // rising edge of "MbPCS1".DONE
   "xPE1P4" := "MbPCS1".DONE;
   IF #_w1 THEN "PCS1".xREQ := FALSE; END_IF;
END_REGION

REGION Network 37: Write RW_Block1 parameter - da controllare password
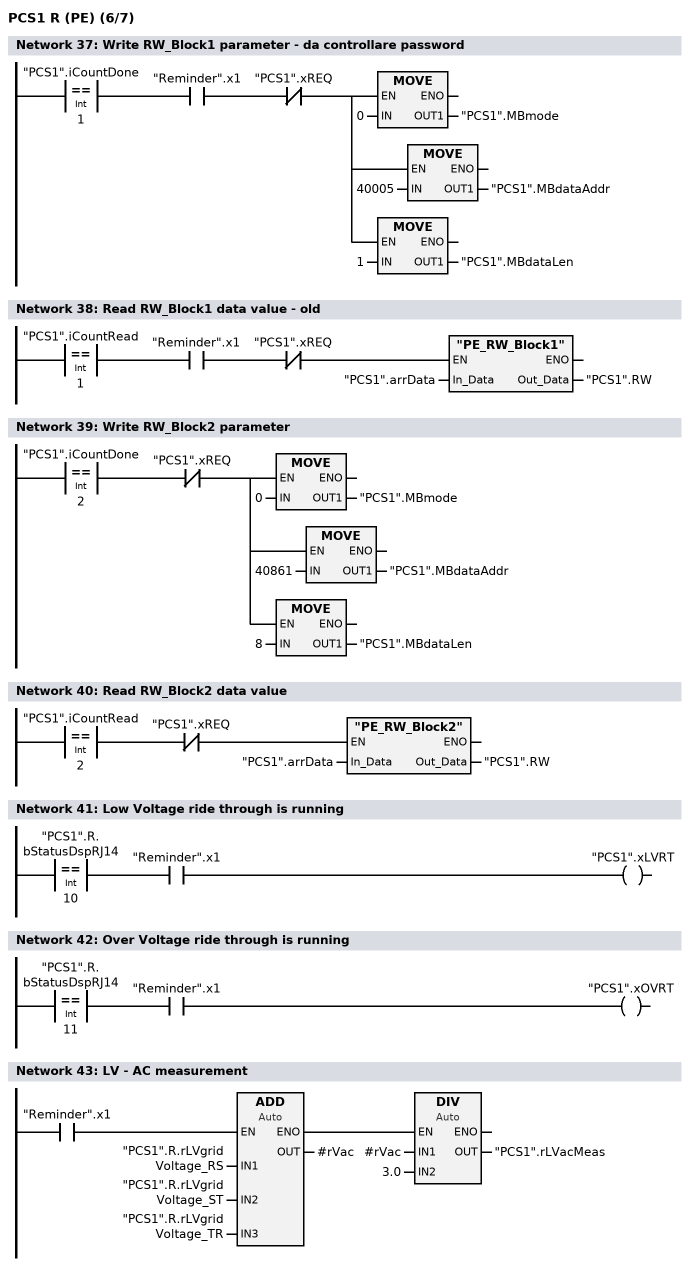
   RUNG wire#powerrail
      { S7_Templates := "SrcType := Int" } EQ_Contact(in1 := "PCS1".iCountDone, in2 := 1)
      Contact( "Reminder".x1 )
      I_Contact( "PCS1".xREQ )
      wire#w1
      Move(in := 0, out1 => "PCS1".MBmode)
   END_RUNG
   RUNG wire#w1
      Move(in := 40005, out1 => "PCS1".MBdataAddr)
   END_RUNG
   RUNG wire#w1
      Move(in := 1, out1 => "PCS1".MBdataLen)
   END_RUNG
   // the same network as SCL:
   IF ("PCS1".iCountDone = 1) AND "Reminder".x1 AND NOT "PCS1".xREQ THEN
       "PCS1".MBmode := 0;
       "PCS1".MBdataAddr := 40005;
       "PCS1".MBdataLen := 1;
   END_IF;
END_REGION

REGION Network 38: Read RW_Block1 data value - old
   RUNG wire#powerrail
      { S7_Templates := "SrcType := Int" } EQ_Contact(in1 := "PCS1".iCountRead, in2 := 1)
      Contact( "Reminder".x1 )
      I_Contact( "PCS1".xREQ )
      "PE_RW_Block1"(In_Data := "PCS1".arrData, Out_Data => "PCS1".RW)
   END_RUNG
   // the same network as SCL:
   IF ("PCS1".iCountRead = 1) AND "Reminder".x1 AND NOT "PCS1".xREQ THEN
       "PE_RW_Block1"(In_Data := "PCS1".arrData, Out_Data => "PCS1".RW);
   END_IF;
END_REGION

REGION Network 39: Write RW_Block2 parameter
   RUNG wire#powerrail
      { S7_Templates := "SrcType := Int" } EQ_Contact(in1 := "PCS1".iCountDone, in2 := 2)
      I_Contact( "PCS1".xREQ )
      wire#w1
      Move(in := 0, out1 => "PCS1".MBmode)
   END_RUNG
   RUNG wire#w1
      Move(in := 40861, out1 => "PCS1".MBdataAddr)
   END_RUNG
   RUNG wire#w1
      Move(in := 8, out1 => "PCS1".MBdataLen)
   END_RUNG
   // the same network as SCL:
   IF ("PCS1".iCountDone = 2) AND NOT "PCS1".xREQ THEN
       "PCS1".MBmode := 0;
       "PCS1".MBdataAddr := 40861;
       "PCS1".MBdataLen := 8;
   END_IF;
END_REGION

REGION Network 40: Read RW_Block2 data value
   RUNG wire#powerrail
      { S7_Templates := "SrcType := Int" } EQ_Contact(in1 := "PCS1".iCountRead, in2 := 2)
      I_Contact( "PCS1".xREQ )
      "PE_RW_Block2"(In_Data := "PCS1".arrData, Out_Data => "PCS1".RW)
   END_RUNG
   // the same network as SCL:
   IF ("PCS1".iCountRead = 2) AND NOT "PCS1".xREQ THEN
       "PE_RW_Block2"(In_Data := "PCS1".arrData, Out_Data => "PCS1".RW);
   END_IF;
END_REGION

REGION Network 41: Low Voltage ride through is running
   RUNG wire#powerrail
      { S7_Templates := "SrcType := Int" } EQ_Contact(in1 := "PCS1".R.bStatusDspRJ14, in2 := 10)
      Contact( "Reminder".x1 )
      Coil( "PCS1".xLVRT )
   END_RUNG
   // the same network as SCL:
   "PCS1".xLVRT := ("PCS1".R.bStatusDspRJ14 = 10) AND "Reminder".x1;
END_REGION

REGION Network 42: Over Voltage ride through is running
   RUNG wire#powerrail
      { S7_Templates := "SrcType := Int" } EQ_Contact(in1 := "PCS1".R.bStatusDspRJ14, in2 := 11)
      Contact( "Reminder".x1 )
      Coil( "PCS1".xOVRT )
   END_RUNG
   // the same network as SCL:
   "PCS1".xOVRT := ("PCS1".R.bStatusDspRJ14 = 11) AND "Reminder".x1;
END_REGION

REGION Network 43: LV - AC measurement
   RUNG wire#powerrail
      Contact( "Reminder".x1 )
      Add(in1 := "PCS1".R.rLVgridVoltage_RS, in2 := "PCS1".R.rLVgridVoltage_ST, in3 := "PCS1".R.rLVgridVoltage_TR, out => #rVac)
      Div(in1 := #rVac, in2 := 3.0, out => "PCS1".rLVacMeas)
   END_RUNG
   // the same network as SCL:
   IF "Reminder".x1 THEN
       #rVac := "PCS1".R.rLVgridVoltage_RS + "PCS1".R.rLVgridVoltage_ST + "PCS1".R.rLVgridVoltage_TR;
       "PCS1".rLVacMeas := #rVac / 3.0;
   END_IF;
END_REGION

REGION Network 44: MV - AC measurement
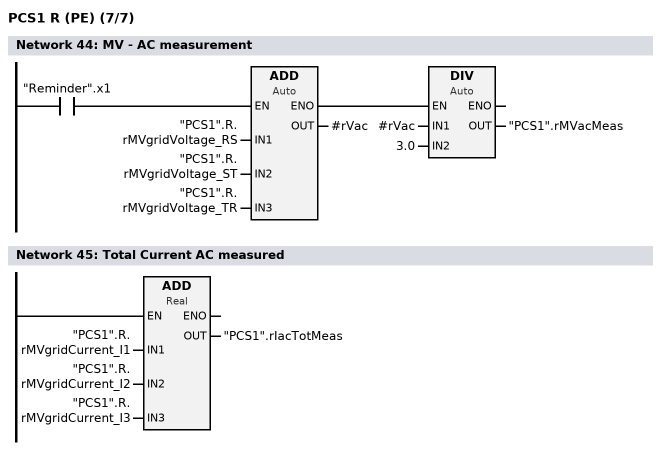
   RUNG wire#powerrail
      Contact( "Reminder".x1 )
      Add(in1 := "PCS1".R.rMVgridVoltage_RS, in2 := "PCS1".R.rMVgridVoltage_ST, in3 := "PCS1".R.rMVgridVoltage_TR, out => #rVac)
      Div(in1 := #rVac, in2 := 3.0, out => "PCS1".rMVacMeas)
   END_RUNG
   // the same network as SCL:
   IF "Reminder".x1 THEN
       #rVac := "PCS1".R.rMVgridVoltage_RS + "PCS1".R.rMVgridVoltage_ST + "PCS1".R.rMVgridVoltage_TR;
       "PCS1".rMVacMeas := #rVac / 3.0;
   END_IF;
END_REGION

REGION Network 45: Total Current AC measured
   RUNG wire#powerrail
      { S7_Templates := "SrcType := Real" } Add(in1 := "PCS1".R.rMVgridCurrent_I1, in2 := "PCS1".R.rMVgridCurrent_I2, in3 := "PCS1".R.rMVgridCurrent_I3, out => "PCS1".rIacTotMeas)
   END_RUNG
   // the same network as SCL:
   "PCS1".rIacTotMeas := "PCS1".R.rMVgridCurrent_I1 + "PCS1".R.rMVgridCurrent_I2 + "PCS1".R.rMVgridCurrent_I3;
END_REGION
END_FUNCTION

FUNCTION "PE_R_41001-41114" : Void
{ S7_Optimized_Access := 'TRUE' }
VERSION : 0.1
   VAR_INPUT 
      Input_Data : Array[1..125] of Word;
   END_VAR

   VAR_OUTPUT 
      Output_Data : "R_PE";
   END_VAR

   VAR_TEMP 
      "DWord" : DWord;
   END_VAR


BEGIN
	
	// 23/03/2023
	REGION
	    #Output_Data.diCurrentFault := WORD_TO_UINT(#Input_Data[1]);
	    #Output_Data.diCurrentFaultModule := WORD_TO_UINT(#Input_Data[2]);
	    #Output_Data.diCurrentWarning := WORD_TO_UINT(#Input_Data[3]);
	    #Output_Data.iCurrentStatus := WORD_TO_INT(#Input_Data[4]);
	    #Output_Data.xStartCondition_f := WORD_TO_BOOL(#Input_Data[41]);
	    #Output_Data.xStartCondition_Vdc := WORD_TO_BOOL(#Input_Data[42]);
	    #Output_Data.xStartCondition_MVcell := WORD_TO_BOOL(#Input_Data[43]);
	    #Output_Data.xStartCondition_P := WORD_TO_BOOL(#Input_Data[44]);
	    #Output_Data.bStatusDspRJ13 := WORD_TO_BYTE(#Input_Data[84]);
	    #Output_Data.bStatusDspRJ14 := WORD_TO_BYTE(#Input_Data[85]);
	    #Output_Data.bStatusDspRJ15 := WORD_TO_BYTE(#Input_Data[86]);
	    #Output_Data.bStatusDspRJ16 := WORD_TO_BYTE(#Input_Data[87]);
	    #Output_Data.bStatusDspRJ20 := WORD_TO_BYTE(#Input_Data[90]);
	    #Output_Data.iMV_PT100_1 := WORD_TO_INT(#Input_Data[109]);
	    #Output_Data.iMV_PT100_2 := WORD_TO_INT(#Input_Data[110]);
	    #Output_Data.iMV_PT100_3 := WORD_TO_INT(#Input_Data[111]);
	    #Output_Data.iP_control := WORD_TO_INT(#Input_Data[113]);
	    #Output_Data.iQ_control := WORD_TO_INT(#Input_Data[114]);
	END_REGION
END_FUNCTION

FUNCTION "PE_R_40632-40640" : Void
{ S7_Optimized_Access := 'TRUE' }
VERSION : 0.1
   VAR_INPUT 
      Input_Data : Array[1..125] of Word;
   END_VAR

   VAR_OUTPUT 
      Output_Data : "R_PE";
   END_VAR

   VAR_TEMP 
      "DWord" : DWord;
   END_VAR


BEGIN
	
	// 23/03/2023
	REGION
	    #Output_Data.iAcSwitchStatus := WORD_TO_INT(#Input_Data[1]);
	    #Output_Data.iMVswitchStatus := WORD_TO_INT(#Input_Data[2]);
	    #Output_Data.iMVgenswitchStatus := WORD_TO_INT(#Input_Data[2]);
	    #Output_Data.iMVearthswitchStatus := WORD_TO_INT(#Input_Data[2]);
	    #Output_Data.iDC1switchStatus := WORD_TO_INT(#Input_Data[2]);
	    #Output_Data.iDC2switchStatus := WORD_TO_INT(#Input_Data[2]);
	    #Output_Data.iDC3switchStatus := WORD_TO_INT(#Input_Data[2]);
	    #Output_Data.iDC4switchStatus := WORD_TO_INT(#Input_Data[44]);
	END_REGION
END_FUNCTION

FUNCTION "PE_R_40928-40930" : Void
{ S7_Optimized_Access := 'TRUE' }
VERSION : 0.1
   VAR_INPUT 
      Input_Data : Array[1..125] of Word;
   END_VAR

   VAR_OUTPUT 
      Output_Data : "R_PE";
   END_VAR

   VAR_TEMP 
      "DWord" : DWord;
   END_VAR


BEGIN
	
	// 23/03/2023
	REGION
	    #Output_Data.xStartCodnition_all := WORD_TO_BOOL(#Input_Data[1]);
	    #Output_Data.xStartCodnition_V := WORD_TO_BOOL(#Input_Data[2]);
	END_REGION
END_FUNCTION

FUNCTION "PE_R_41373-41393" : Void
{ S7_Optimized_Access := 'TRUE' }
VERSION : 0.1
   VAR_INPUT 
      Input_Data : Array[1..125] of Word;
   END_VAR

   VAR_OUTPUT 
      Output_Data : "R_PE";
   END_VAR

   VAR_TEMP 
      "DWord" : DWord;
   END_VAR


BEGIN
	
	// 23/03/2023
	REGION
	    #Output_Data.iInputPower_1 := WORD_TO_INT(#Input_Data[1]);
	    #Output_Data.iInputPower_2 := WORD_TO_INT(#Input_Data[2]);
	    #Output_Data.iInputPower_3 := WORD_TO_INT(#Input_Data[3]);
	    #Output_Data.iInputPower_4 := WORD_TO_INT(#Input_Data[4]);
	    #Output_Data.rI_DC1 := INT_TO_REAL(WORD_TO_INT(#Input_Data[5]));
	    #Output_Data.rI_DC2 := INT_TO_REAL(WORD_TO_INT(#Input_Data[6]));
	    #Output_Data.rI_DC3 := INT_TO_REAL(WORD_TO_INT(#Input_Data[7]));
	    #Output_Data.rI_DC4 := INT_TO_REAL(WORD_TO_INT(#Input_Data[8]));
	    #Output_Data.rDCvoltageBus_1 := INT_TO_REAL(WORD_TO_INT(#Input_Data[9]));
	    #Output_Data.rDCvoltageBus_2 := INT_TO_REAL(WORD_TO_INT(#Input_Data[10]));
	    #Output_Data.rDCvoltageBus_3 := INT_TO_REAL(WORD_TO_INT(#Input_Data[11]));
	    #Output_Data.rDCvoltageBus_4 := INT_TO_REAL(WORD_TO_INT(#Input_Data[12]));
	    #Output_Data.rDCvoltageExt_1 := INT_TO_REAL(WORD_TO_INT(#Input_Data[13]));
	    #Output_Data.rDCvoltageExt_2 := INT_TO_REAL(WORD_TO_INT(#Input_Data[14]));
	    #Output_Data.rDCvoltageExt_3 := INT_TO_REAL(WORD_TO_INT(#Input_Data[15]));
	    #Output_Data.rDCvoltageExt_4 := INT_TO_REAL(WORD_TO_INT(#Input_Data[16]));
	    #Output_Data.rDCvoltageLast_1 := INT_TO_REAL(WORD_TO_INT(#Input_Data[17]));
	    #Output_Data.rDCvoltageLast_2 := INT_TO_REAL(WORD_TO_INT(#Input_Data[18]));
	    #Output_Data.rDCvoltageLast_3 := INT_TO_REAL(WORD_TO_INT(#Input_Data[19]));
	    #Output_Data.rDCvoltageLast_4 := INT_TO_REAL(WORD_TO_INT(#Input_Data[20]));
	END_REGION
END_FUNCTION

FUNCTION "PE_R_44301-44323" : Void
{ S7_Optimized_Access := 'TRUE' }
VERSION : 0.1
   VAR_INPUT 
      Input_Data : Array[1..125] of Word;
   END_VAR

   VAR_OUTPUT 
      Output_Data : "R_PE";
   END_VAR

   VAR_TEMP 
      "DWord" : DWord;
   END_VAR


BEGIN
	
	// 23/03/2023
	REGION
	    #Output_Data.rMVgridVoltage_RS := INT_TO_REAL(WORD_TO_INT(#Input_Data[1]));
	    #Output_Data.rMVgridVoltage_ST := INT_TO_REAL(WORD_TO_INT(#Input_Data[2]));
	    #Output_Data.rMVgridVoltage_TR := INT_TO_REAL(WORD_TO_INT(#Input_Data[3]));
	    #Output_Data.rMVgridCurrent_I1 := INT_TO_REAL(WORD_TO_INT(#Input_Data[4]));
	    #Output_Data.rMVgridCurrent_I2 := INT_TO_REAL(WORD_TO_INT(#Input_Data[5]));
	    #Output_Data.rMVgridCurrent_I3 := INT_TO_REAL(WORD_TO_INT(#Input_Data[6]));
	    #Output_Data.iMV_P := WORD_TO_INT(#Input_Data[7]);
	    #Output_Data.iMV_Q := WORD_TO_INT(#Input_Data[8]);
	    #Output_Data.uiMV_S := WORD_TO_UINT(#Input_Data[9]);
	    #Output_Data.rMVcosphi := INT_TO_REAL(WORD_TO_INT(#Input_Data[10]));
	    #Output_Data.rLVgridVoltage_RS := INT_TO_REAL(WORD_TO_INT(#Input_Data[11]));
	    #Output_Data.rLVgridVoltage_ST := INT_TO_REAL(WORD_TO_INT(#Input_Data[12]));
	    #Output_Data.rLVgridVoltage_TR := INT_TO_REAL(WORD_TO_INT(#Input_Data[13]));
	    #Output_Data.rLVgridCurrent_I1 := INT_TO_REAL(WORD_TO_INT(#Input_Data[14]));
	    #Output_Data.rLVgridCurrent_I2 := INT_TO_REAL(WORD_TO_INT(#Input_Data[15]));
	    #Output_Data.rLVgridCurrent_I3 := INT_TO_REAL(WORD_TO_INT(#Input_Data[16]));
	    #Output_Data.iLV_P := WORD_TO_INT(#Input_Data[17]);
	    #Output_Data.iLV_Q := WORD_TO_INT(#Input_Data[18]);
	    #Output_Data.uiLV_S := WORD_TO_UINT(#Input_Data[19]);
	    #Output_Data.rLVcosphi := INT_TO_REAL(WORD_TO_INT(#Input_Data[20]));
	    #Output_Data.xGridSequency := WORD_TO_BOOL(#Input_Data[21]);
	    #Output_Data.rGridFreq := INT_TO_REAL(WORD_TO_INT(#Input_Data[22]));
	END_REGION
END_FUNCTION

FUNCTION "PE_R_Module_1" : Void
{ S7_Optimized_Access := 'TRUE' }
VERSION : 0.1
   VAR_INPUT 
      Input_Data : Array[1..125] of Word;
   END_VAR

   VAR_OUTPUT 
      Output_Data : "R_PE";
   END_VAR

   VAR_TEMP 
      "DWord" : DWord;
   END_VAR


BEGIN
	
	// 23/03/2023
	REGION
	    #Output_Data.Module_1.bModuleStatus := #Input_Data[1];
	    #Output_Data.Module_1.rCurrent_R := INT_TO_REAL(WORD_TO_INT(#Input_Data[2]));
	    #Output_Data.Module_1.rCurrent_S := INT_TO_REAL(WORD_TO_INT(#Input_Data[3]));
	    #Output_Data.Module_1.rCurrent_T := INT_TO_REAL(WORD_TO_INT(#Input_Data[4]));
	    #Output_Data.Module_1.rDC_current := INT_TO_REAL(WORD_TO_INT(#Input_Data[5]));
	    #Output_Data.Module_1.iDC_voltage_P := WORD_TO_INT(#Input_Data[6]);
	    #Output_Data.Module_1.iDC_voltage_N := WORD_TO_INT(#Input_Data[7]);
	    #Output_Data.Module_1.iDC_voltage := WORD_TO_INT(#Input_Data[8]);
	    #Output_Data.Module_1.rActivePower := INT_TO_REAL(WORD_TO_INT(#Input_Data[9]));
	    #Output_Data.Module_1.rReactivePower := INT_TO_REAL(WORD_TO_INT(#Input_Data[10]));
	    #Output_Data.Module_1.uiAC_voltage_R := WORD_TO_UINT(#Input_Data[11]);
	    #Output_Data.Module_1.uiAC_voltage_S := WORD_TO_UINT(#Input_Data[12]);
	    #Output_Data.Module_1.uiAC_voltage_T := WORD_TO_UINT(#Input_Data[13]);
	    #Output_Data.Module_1.iAmbientTemperature := WORD_TO_INT(#Input_Data[14]);
	    #Output_Data.Module_1.iMaxTemperature := WORD_TO_INT(#Input_Data[15]);
	    #Output_Data.Module_1.usiHumidity := WORD_TO_USINT(#Input_Data[16]);
	END_REGION
END_FUNCTION

FUNCTION "PE_R_Module_2" : Void
{ S7_Optimized_Access := 'TRUE' }
VERSION : 0.1
   VAR_INPUT 
      Input_Data : Array[1..125] of Word;
   END_VAR

   VAR_OUTPUT 
      Output_Data : "R_PE";
   END_VAR

   VAR_TEMP 
      "DWord" : DWord;
   END_VAR


BEGIN
	
	// 23/03/2023
	REGION
	    #Output_Data.Module_2.bModuleStatus := #Input_Data[1];
	    #Output_Data.Module_2.rCurrent_R := INT_TO_REAL(WORD_TO_INT(#Input_Data[2]));
	    #Output_Data.Module_2.rCurrent_S := INT_TO_REAL(WORD_TO_INT(#Input_Data[3]));
	    #Output_Data.Module_2.rCurrent_T := INT_TO_REAL(WORD_TO_INT(#Input_Data[4]));
	    #Output_Data.Module_2.rDC_current := INT_TO_REAL(WORD_TO_INT(#Input_Data[5]));
	    #Output_Data.Module_2.iDC_voltage_P := WORD_TO_INT(#Input_Data[6]);
	    #Output_Data.Module_2.iDC_voltage_N := WORD_TO_INT(#Input_Data[7]);
	    #Output_Data.Module_2.iDC_voltage := WORD_TO_INT(#Input_Data[8]);
	    #Output_Data.Module_2.rActivePower := INT_TO_REAL(WORD_TO_INT(#Input_Data[9]));
	    #Output_Data.Module_2.rReactivePower := INT_TO_REAL(WORD_TO_INT(#Input_Data[10]));
	    #Output_Data.Module_2.uiAC_voltage_R := WORD_TO_UINT(#Input_Data[11]);
	    #Output_Data.Module_2.uiAC_voltage_S := WORD_TO_UINT(#Input_Data[12]);
	    #Output_Data.Module_2.uiAC_voltage_T := WORD_TO_UINT(#Input_Data[13]);
	    #Output_Data.Module_2.iAmbientTemperature := WORD_TO_INT(#Input_Data[14]);
	    #Output_Data.Module_2.iMaxTemperature := WORD_TO_INT(#Input_Data[15]);
	    #Output_Data.Module_2.usiHumidity := WORD_TO_USINT(#Input_Data[16]);
	END_REGION
END_FUNCTION

FUNCTION "PE_R_Module_3" : Void
{ S7_Optimized_Access := 'TRUE' }
VERSION : 0.1
   VAR_INPUT 
      Input_Data : Array[1..125] of Word;
   END_VAR

   VAR_OUTPUT 
      Output_Data : "R_PE";
   END_VAR

   VAR_TEMP 
      "DWord" : DWord;
   END_VAR


BEGIN
	
	// 23/03/2023
	REGION
	    #Output_Data.Module_3.bModuleStatus := #Input_Data[1];
	    #Output_Data.Module_3.rCurrent_R := INT_TO_REAL(WORD_TO_INT(#Input_Data[2]));
	    #Output_Data.Module_3.rCurrent_S := INT_TO_REAL(WORD_TO_INT(#Input_Data[3]));
	    #Output_Data.Module_3.rCurrent_T := INT_TO_REAL(WORD_TO_INT(#Input_Data[4]));
	    #Output_Data.Module_3.rDC_current := INT_TO_REAL(WORD_TO_INT(#Input_Data[5]));
	    #Output_Data.Module_3.iDC_voltage_P := WORD_TO_INT(#Input_Data[6]);
	    #Output_Data.Module_3.iDC_voltage_N := WORD_TO_INT(#Input_Data[7]);
	    #Output_Data.Module_3.iDC_voltage := WORD_TO_INT(#Input_Data[8]);
	    #Output_Data.Module_3.rActivePower := INT_TO_REAL(WORD_TO_INT(#Input_Data[9]));
	    #Output_Data.Module_3.rReactivePower := INT_TO_REAL(WORD_TO_INT(#Input_Data[10]));
	    #Output_Data.Module_3.uiAC_voltage_R := WORD_TO_UINT(#Input_Data[11]);
	    #Output_Data.Module_3.uiAC_voltage_S := WORD_TO_UINT(#Input_Data[12]);
	    #Output_Data.Module_3.uiAC_voltage_T := WORD_TO_UINT(#Input_Data[13]);
	    #Output_Data.Module_3.iAmbientTemperature := WORD_TO_INT(#Input_Data[14]);
	    #Output_Data.Module_3.iMaxTemperature := WORD_TO_INT(#Input_Data[15]);
	    #Output_Data.Module_3.usiHumidity := WORD_TO_USINT(#Input_Data[16]);
	END_REGION
END_FUNCTION

FUNCTION "PE_R_Module_4" : Void
{ S7_Optimized_Access := 'TRUE' }
VERSION : 0.1
   VAR_INPUT 
      Input_Data : Array[1..125] of Word;
   END_VAR

   VAR_OUTPUT 
      Output_Data : "R_PE";
   END_VAR

   VAR_TEMP 
      "DWord" : DWord;
   END_VAR


BEGIN
	
	// 23/03/2023
	REGION
	    #Output_Data.Module_4.bModuleStatus := #Input_Data[1];
	    #Output_Data.Module_4.rCurrent_R := INT_TO_REAL(WORD_TO_INT(#Input_Data[2]));
	    #Output_Data.Module_4.rCurrent_S := INT_TO_REAL(WORD_TO_INT(#Input_Data[3]));
	    #Output_Data.Module_4.rCurrent_T := INT_TO_REAL(WORD_TO_INT(#Input_Data[4]));
	    #Output_Data.Module_4.rDC_current := INT_TO_REAL(WORD_TO_INT(#Input_Data[5]));
	    #Output_Data.Module_4.iDC_voltage_P := WORD_TO_INT(#Input_Data[6]);
	    #Output_Data.Module_4.iDC_voltage_N := WORD_TO_INT(#Input_Data[7]);
	    #Output_Data.Module_4.iDC_voltage := WORD_TO_INT(#Input_Data[8]);
	    #Output_Data.Module_4.rActivePower := INT_TO_REAL(WORD_TO_INT(#Input_Data[9]));
	    #Output_Data.Module_4.rReactivePower := INT_TO_REAL(WORD_TO_INT(#Input_Data[10]));
	    #Output_Data.Module_4.uiAC_voltage_R := WORD_TO_UINT(#Input_Data[11]);
	    #Output_Data.Module_4.uiAC_voltage_S := WORD_TO_UINT(#Input_Data[12]);
	    #Output_Data.Module_4.uiAC_voltage_T := WORD_TO_UINT(#Input_Data[13]);
	    #Output_Data.Module_4.iAmbientTemperature := WORD_TO_INT(#Input_Data[14]);
	    #Output_Data.Module_4.iMaxTemperature := WORD_TO_INT(#Input_Data[15]);
	    #Output_Data.Module_4.usiHumidity := WORD_TO_USINT(#Input_Data[16]);
	END_REGION
END_FUNCTION

FUNCTION "PE_R_Humidity" : Void
{ S7_Optimized_Access := 'TRUE' }
VERSION : 0.1
   VAR_INPUT 
      Input_Data : Array[1..125] of Word;
   END_VAR

   VAR_OUTPUT 
      Output_Data : "R_PE";
   END_VAR

   VAR_TEMP 
      "DWord" : DWord;
   END_VAR


BEGIN
	
	// 23/03/2023
	REGION
	    #Output_Data.Module_1.usiHumidity := WORD_TO_USINT(#Input_Data[1]);
	    #Output_Data.Module_2.usiHumidity := WORD_TO_USINT(#Input_Data[2]);
	    #Output_Data.Module_3.usiHumidity := WORD_TO_USINT(#Input_Data[3]);
	    #Output_Data.Module_4.usiHumidity := WORD_TO_USINT(#Input_Data[4]);
	END_REGION
END_FUNCTION

FUNCTION "PCS1 R (S)" : Void   // FC43, LAD
TITLE = ModBus TCP for PCS Power Electronics
{ S7_Optimized_Access := 'TRUE' }
VERSION : 0.1
// stored: AutoNumber false, IsIECCheckEnabled false, SetENOAutomatically false, UDAEnableTagReadback false
   VAR_TEMP
      rVac : Real;
   END_VAR
   VAR_TEMP   // added for the SCL form of the ladder/FBD networks
      _w1 : Bool;
   END_VAR
BEGIN

REGION Network 1: Function Modbus Client
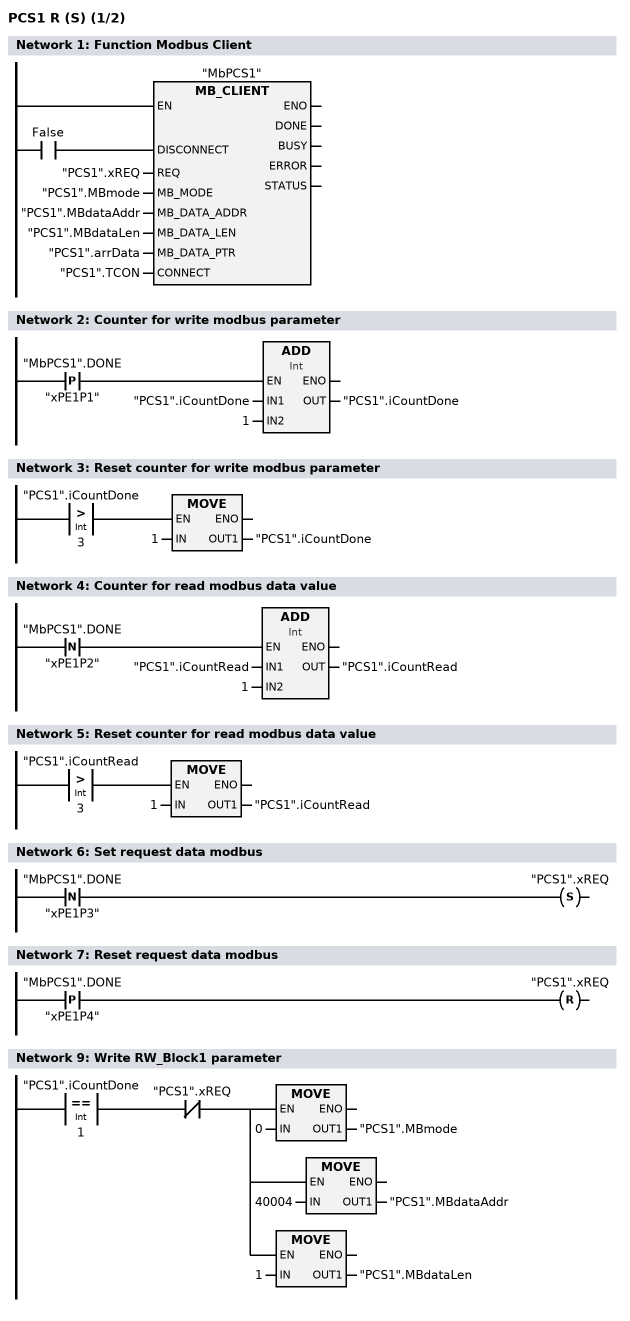
   RUNG wire#powerrail
      "MbPCS1".MB_CLIENT(DISCONNECT := wire#w1, REQ := "PCS1".xREQ, MB_MODE := "PCS1".MBmode, MB_DATA_ADDR := "PCS1".MBdataAddr, MB_DATA_LEN := "PCS1".MBdataLen, MB_DATA_PTR := "PCS1".arrData, CONNECT := "PCS1".TCON, DONE =>, BUSY =>, ERROR =>, STATUS =>)
   END_RUNG
   RUNG wire#powerrail
      Contact( False )
   END_RUNG wire#w1
   // the same network as SCL:
   "MbPCS1"(DISCONNECT := False,   // MB_CLIENT
            REQ := "PCS1".xREQ,
            MB_MODE := "PCS1".MBmode,
            MB_DATA_ADDR := "PCS1".MBdataAddr,
            MB_DATA_LEN := "PCS1".MBdataLen,
            MB_DATA_PTR := "PCS1".arrData,
            CONNECT := "PCS1".TCON);
END_REGION

REGION Network 2: Counter for write modbus parameter
   RUNG wire#powerrail
      P_Contact(operand := "MbPCS1".DONE, bit := "xPE1P1")
      { S7_Templates := "SrcType := Int" } Add(in1 := "PCS1".iCountDone, in2 := 1, out => "PCS1".iCountDone)
   END_RUNG
   // the same network as SCL:
   #_w1 := "MbPCS1".DONE AND NOT "xPE1P1";   // rising edge of "MbPCS1".DONE
   "xPE1P1" := "MbPCS1".DONE;
   IF #_w1 THEN "PCS1".iCountDone := "PCS1".iCountDone + 1; END_IF;
END_REGION

REGION Network 3: Reset counter for write modbus parameter
   RUNG wire#powerrail
      { S7_Templates := "SrcType := Int" } GT_Contact(in1 := "PCS1".iCountDone, in2 := 3)
      Move(in := 1, out1 => "PCS1".iCountDone)
   END_RUNG
   // the same network as SCL:
   IF "PCS1".iCountDone > 3 THEN "PCS1".iCountDone := 1; END_IF;
END_REGION

REGION Network 4: Counter for read modbus data value
   RUNG wire#powerrail
      N_Contact(operand := "MbPCS1".DONE, bit := "xPE1P2")
      { S7_Templates := "SrcType := Int" } Add(in1 := "PCS1".iCountRead, in2 := 1, out => "PCS1".iCountRead)
   END_RUNG
   // the same network as SCL:
   #_w1 := NOT "MbPCS1".DONE AND "xPE1P2";   // falling edge of "MbPCS1".DONE
   "xPE1P2" := "MbPCS1".DONE;
   IF #_w1 THEN "PCS1".iCountRead := "PCS1".iCountRead + 1; END_IF;
END_REGION

REGION Network 5: Reset counter for read modbus data value
   RUNG wire#powerrail
      { S7_Templates := "SrcType := Int" } GT_Contact(in1 := "PCS1".iCountRead, in2 := 3)
      Move(in := 1, out1 => "PCS1".iCountRead)
   END_RUNG
   // the same network as SCL:
   IF "PCS1".iCountRead > 3 THEN "PCS1".iCountRead := 1; END_IF;
END_REGION

REGION Network 6: Set request data modbus
   RUNG wire#powerrail
      N_Contact(operand := "MbPCS1".DONE, bit := "xPE1P3")
      S_Coil( "PCS1".xREQ )
   END_RUNG
   // the same network as SCL:
   #_w1 := NOT "MbPCS1".DONE AND "xPE1P3";   // falling edge of "MbPCS1".DONE
   "xPE1P3" := "MbPCS1".DONE;
   IF #_w1 THEN "PCS1".xREQ := TRUE; END_IF;
END_REGION

REGION Network 7: Reset request data modbus
   RUNG wire#powerrail
      P_Contact(operand := "MbPCS1".DONE, bit := "xPE1P4")
      R_Coil( "PCS1".xREQ )
   END_RUNG
   // the same network as SCL:
   #_w1 := "MbPCS1".DONE AND NOT "xPE1P4";   // rising edge of "MbPCS1".DONE
   "xPE1P4" := "MbPCS1".DONE;
   IF #_w1 THEN "PCS1".xREQ := FALSE; END_IF;
END_REGION

REGION Network 9: Write RW_Block1 parameter
   RUNG wire#powerrail
      { S7_Templates := "SrcType := Int" } EQ_Contact(in1 := "PCS1".iCountDone, in2 := 1)
      I_Contact( "PCS1".xREQ )
      wire#w1
      Move(in := 0, out1 => "PCS1".MBmode)
   END_RUNG
   RUNG wire#w1
      Move(in := 40004, out1 => "PCS1".MBdataAddr)
   END_RUNG
   RUNG wire#w1
      Move(in := 1, out1 => "PCS1".MBdataLen)
   END_RUNG
   // the same network as SCL:
   IF ("PCS1".iCountDone = 1) AND NOT "PCS1".xREQ THEN
       "PCS1".MBmode := 0;
       "PCS1".MBdataAddr := 40004;
       "PCS1".MBdataLen := 1;
   END_IF;
END_REGION

REGION Network 10: Read RW_Block1 data value
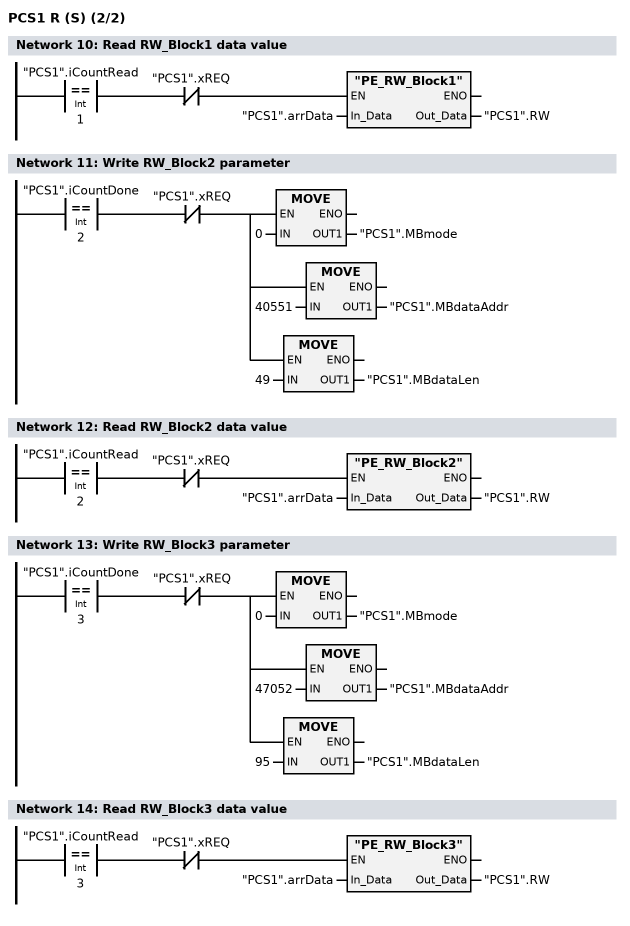
   RUNG wire#powerrail
      { S7_Templates := "SrcType := Int" } EQ_Contact(in1 := "PCS1".iCountRead, in2 := 1)
      I_Contact( "PCS1".xREQ )
      "PE_RW_Block1"(In_Data := "PCS1".arrData, Out_Data => "PCS1".RW)
   END_RUNG
   // the same network as SCL:
   IF ("PCS1".iCountRead = 1) AND NOT "PCS1".xREQ THEN
       "PE_RW_Block1"(In_Data := "PCS1".arrData, Out_Data => "PCS1".RW);
   END_IF;
END_REGION

REGION Network 11: Write RW_Block2 parameter
   RUNG wire#powerrail
      { S7_Templates := "SrcType := Int" } EQ_Contact(in1 := "PCS1".iCountDone, in2 := 2)
      I_Contact( "PCS1".xREQ )
      wire#w1
      Move(in := 0, out1 => "PCS1".MBmode)
   END_RUNG
   RUNG wire#w1
      Move(in := 40551, out1 => "PCS1".MBdataAddr)
   END_RUNG
   RUNG wire#w1
      Move(in := 49, out1 => "PCS1".MBdataLen)
   END_RUNG
   // the same network as SCL:
   IF ("PCS1".iCountDone = 2) AND NOT "PCS1".xREQ THEN
       "PCS1".MBmode := 0;
       "PCS1".MBdataAddr := 40551;
       "PCS1".MBdataLen := 49;
   END_IF;
END_REGION

REGION Network 12: Read RW_Block2 data value
   RUNG wire#powerrail
      { S7_Templates := "SrcType := Int" } EQ_Contact(in1 := "PCS1".iCountRead, in2 := 2)
      I_Contact( "PCS1".xREQ )
      "PE_RW_Block2"(In_Data := "PCS1".arrData, Out_Data => "PCS1".RW)
   END_RUNG
   // the same network as SCL:
   IF ("PCS1".iCountRead = 2) AND NOT "PCS1".xREQ THEN
       "PE_RW_Block2"(In_Data := "PCS1".arrData, Out_Data => "PCS1".RW);
   END_IF;
END_REGION

REGION Network 13: Write RW_Block3 parameter
   RUNG wire#powerrail
      { S7_Templates := "SrcType := Int" } EQ_Contact(in1 := "PCS1".iCountDone, in2 := 3)
      I_Contact( "PCS1".xREQ )
      wire#w1
      Move(in := 0, out1 => "PCS1".MBmode)
   END_RUNG
   RUNG wire#w1
      Move(in := 47052, out1 => "PCS1".MBdataAddr)
   END_RUNG
   RUNG wire#w1
      Move(in := 95, out1 => "PCS1".MBdataLen)
   END_RUNG
   // the same network as SCL:
   IF ("PCS1".iCountDone = 3) AND NOT "PCS1".xREQ THEN
       "PCS1".MBmode := 0;
       "PCS1".MBdataAddr := 47052;
       "PCS1".MBdataLen := 95;
   END_IF;
END_REGION

REGION Network 14: Read RW_Block3 data value
   RUNG wire#powerrail
      { S7_Templates := "SrcType := Int" } EQ_Contact(in1 := "PCS1".iCountRead, in2 := 3)
      I_Contact( "PCS1".xREQ )
      "PE_RW_Block3"(In_Data := "PCS1".arrData, Out_Data => "PCS1".RW)
   END_RUNG
   // the same network as SCL:
   IF ("PCS1".iCountRead = 3) AND NOT "PCS1".xREQ THEN
       "PE_RW_Block3"(In_Data := "PCS1".arrData, Out_Data => "PCS1".RW);
   END_IF;
END_REGION
END_FUNCTION

FUNCTION "PE_RW_Block3" : Void
{ S7_Optimized_Access := 'TRUE' }
VERSION : 0.1
   VAR_INPUT 
      In_Data : Array[1..125] of Word;   // pcs
   END_VAR

   VAR_OUTPUT 
      Out_Data : "RW_PE";
   END_VAR


BEGIN
	REGION
	    // 2022/01/24
	END_REGION
	
	REGION
	    
	    //#Out_Data.wBankDcEnbCmd := #In_Data[1];
	    //#Out_Data.rPac1Ref      := INT_TO_REAL(WORD_TO_INT(#In_Data[94]))/100.0;
	    //#Out_Data.rPac2Ref      := INT_TO_REAL(WORD_TO_INT(#In_Data[95]))/100.0;
	    
	END_REGION
END_FUNCTION

FUNCTION "PCS1 W (PE)" : Void   // FC42, LAD
TITLE = ModBus TCP for PCS Power Electronics
{ S7_Optimized_Access := 'TRUE' }
VERSION : 0.1
// stored: AutoNumber false, IsIECCheckEnabled false, SetENOAutomatically false, UDAEnableTagReadback false
   VAR_TEMP
      rSS1PacRef : Real;
      rSS2PacRef : Real;
      rSS1QacRef : Real;
      rSS2QacRef : Real;
      rSnHalfPE : Real;
   END_VAR
   VAR_TEMP   // added for the SCL form of the ladder/FBD networks
      _w1 : Bool;
      _w2 : Bool;
   END_VAR
BEGIN

REGION Network 1: Function Modbus Client
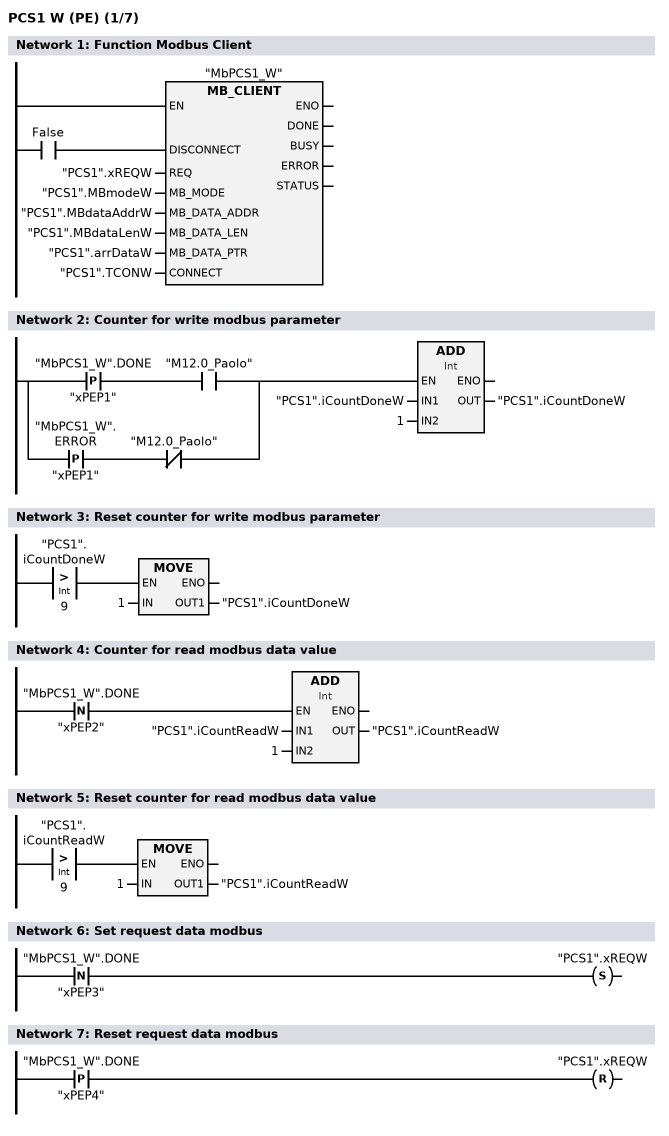
   RUNG wire#powerrail
      "MbPCS1_W".MB_CLIENT(DISCONNECT := wire#w1, REQ := "PCS1".xREQW, MB_MODE := "PCS1".MBmodeW, MB_DATA_ADDR := "PCS1".MBdataAddrW, MB_DATA_LEN := "PCS1".MBdataLenW, MB_DATA_PTR := "PCS1".arrDataW, CONNECT := "PCS1".TCONW, DONE =>, BUSY =>, ERROR =>, STATUS =>)
   END_RUNG
   RUNG wire#powerrail
      Contact( False )
   END_RUNG wire#w1
   // the same network as SCL:
   "MbPCS1_W"(DISCONNECT := False,   // MB_CLIENT
              REQ := "PCS1".xREQW,
              MB_MODE := "PCS1".MBmodeW,
              MB_DATA_ADDR := "PCS1".MBdataAddrW,
              MB_DATA_LEN := "PCS1".MBdataLenW,
              MB_DATA_PTR := "PCS1".arrDataW,
              CONNECT := "PCS1".TCONW);
END_REGION

REGION Network 2: Counter for write modbus parameter
   RUNG wire#powerrail
      P_Contact(operand := "MbPCS1_W".DONE, bit := "xPEP1")
      Contact( "M12.0_Paolo" )
      wire#w1
      { S7_Templates := "SrcType := Int" } Add(in1 := "PCS1".iCountDoneW, in2 := 1, out => "PCS1".iCountDoneW)
   END_RUNG
   RUNG wire#powerrail
      P_Contact(operand := "MbPCS1_W".ERROR, bit := "xPEP1")
      I_Contact( "M12.0_Paolo" )
   END_RUNG wire#w1
   // the same network as SCL:
   #_w1 := "MbPCS1_W".DONE AND NOT "xPEP1";   // rising edge of "MbPCS1_W".DONE
   "xPEP1" := "MbPCS1_W".DONE;
   #_w2 := "MbPCS1_W".ERROR AND NOT "xPEP1";   // rising edge of "MbPCS1_W".ERROR
   "xPEP1" := "MbPCS1_W".ERROR;
   IF (#_w1 AND "M12.0_Paolo") OR (#_w2 AND NOT "M12.0_Paolo") THEN
       "PCS1".iCountDoneW := "PCS1".iCountDoneW + 1;
   END_IF;
END_REGION

